C01819=1046.812,379.525,376.002,173.658,41.858,158.138
C01820=1046.820,379.771,375.961,173.664,41.863,158.140
C01821=1046.829,380.018,375.920,173.671,41.869,158.141
C01822=1046.836,380.264,375.878,173.677,41.874,158.143
C01823=1046.844,380.510,375.838,173.684,41.880,158.145
C01824=1046.852,380.757,375.797,173.690,41.885,158.146
C01825=1046.861,381.004,375.756,173.697,41.890,158.148
C01826=1046.869,381.250,375.714,173.703,41.896,158.150
C01827=1046.877,381.496,375.673,173.710,41.901,158.152
C01828=1046.885,381.743,375.632,173.716,41.907,158.154
C01829=1046.893,381.989,375.590,173.723,41.912,158.155
C01830=1046.901,382.236,375.549,173.729,41.917,158.157
C01831=1046.910,382.481,375.508,173.737,41.923,158.159
C01832=1046.918,382.728,375.467,173.743,41.929,158.161
C01833=1046.926,382.974,375.425,173.750,41.934,158.162
C01834=1046.934,383.221,375.385,173.757,41.939,158.164
C01835=1046.943,383.467,375.343,173.763,41.945,158.166
C01836=1046.950,383.714,375.302,173.770,41.950,158.168
C01837=1046.959,383.960,375.260,173.777,41.956,158.170
C01838=1046.967,384.206,375.219,173.784,41.962,158.171
C01839=1046.975,384.453,375.177,173.791,41.967,158.173
C01840=1046.984,384.699,375.136,173.797,41.973,158.175
C01841=1046.993,384.945,375.094,173.804,41.978,158.177
C01842=1047.001,385.191,375.053,173.811,41.984,158.179
C01843=1047.009,385.438,375.011,173.818,41.989,158.180
C01844=1047.018,385.684,374.969,173.825,41.995,158.182
C01845=1047.026,385.930,374.928,173.832,42.001,158.184
C01846=1047.034,386.177,374.886,173.839,42.006,158.186
C01847=1047.043,386.424,374.845,173.845,42.012,158.188
C01848=1047.051,386.669,374.803,173.852,42.018,158.190
C01849=1047.059,386.916,374.761,173.860,42.023,158.192
C01850=1047.068,387.162,374.719,173.867,42.029,158.193
C01851=1047.076,387.408,374.677,173.873,42.035,158.195
C01852=1047.085,387.655,374.635,173.880,42.041,158.197
C01853=1047.094,387.901,374.594,173.888,42.046,158.199
C01854=1047.102,388.147,374.551,173.895,42.052,158.201
C01855=1047.111,388.393,374.509,173.902,42.058,158.203
C01856=1047.120,388.639,374.468,173.909,42.064,158.205
C01857=1047.128,388.886,374.425,173.916,42.069,158.207
C01858=1047.137,389.132,374.384,173.923,42.075,158.209
C01859=1047.145,389.378,374.341,173.930,42.081,158.210
C01860=1047.158,389.751,374.278,173.941,42.090,158.213
C01861=1047.170,390.124,374.213,173.953,42.099,158.216
C01862=1047.184,390.498,374.149,173.963,42.108,158.219
C01863=1047.196,390.871,374.085,173.974,42.117,158.222
C01864=1047.205,391.117,374.042,173.981,42.123,158.224
C01865=1047.214,391.364,374.000,173.988,42.129,158.226
C01866=1047.222,391.610,373.957,173.996,42.135,158.228
C01867=1047.231,391.856,373.915,174.003,42.141,158.230
C01868=1047.240,392.102,373.872,174.011,42.147,158.232
C01869=1047.248,392.348,373.829,174.018,42.153,158.234
C01870=1047.256,392.595,373.787,174.026,42.160,158.236
C01871=1047.266,392.841,373.744,174.033,42.166,158.238
C01872=1047.274,393.087,373.701,174.041,42.172,158.240
C01873=1047.283,393.333,373.658,174.048,42.178,158.242
C01874=1047.291,393.579,373.615,174.055,42.184,158.244
C01875=1047.300,393.825,373.572,174.063,42.190,158.247
C01876=1047.308,394.071,373.531,174.071,42.196,158.249
C01877=1047.317,394.317,373.487,174.078,42.202,158.251
C01878=1047.325,394.563,373.444,174.086,42.209,158.253
C01879=1047.334,394.809,373.401,174.093,42.215,158.255
C01880=1047.343,395.055,373.359,174.100,42.221,158.257
C01881=1047.352,395.300,373.315,174.108,42.228,158.259
C01882=1047.361,395.547,373.272,174.116,42.234,158.261
C01883=1047.370,395.793,373.229,174.123,42.240,158.263
C01884=1047.378,396.039,373.186,174.131,42.247,158.265
C01885=1047.387,396.285,373.143,174.138,42.253,158.267
C01886=1047.395,396.531,373.100,174.146,42.259,158.270
C01887=1047.404,396.777,373.056,174.154,42.266,158.272
C01888=1047.413,397.024,373.013,174.161,42.272,158.274
C01889=1047.422,397.270,372.970,174.170,42.278,158.276
C01890=1047.430,397.515,372.926,174.177,42.285,158.278
C01891=1047.439,397.761,372.883,174.185,42.291,158.280
C01892=1047.448,398.007,372.839,174.193,42.298,158.282
C01893=1047.457,398.253,372.796,174.200,42.304,158.285
C01894=1047.466,398.499,372.752,174.208,42.311,158.287
C01895=1047.475,398.746,372.709,174.217,42.317,158.289
C01896=1047.483,398.991,372.665,174.224,42.324,158.291
C01897=1047.492,399.236,372.621,174.232,42.330,158.293
C01898=1047.501,399.483,372.578,174.240,42.337,158.296
C01899=1047.510,399.729,372.534,174.248,42.343,158.298
C01900=1047.520,399.975,372.490,174.256,42.350,158.300
C01901=1047.528,400.221,372.447,174.264,42.357,158.302
C01902=1047.538,400.467,372.403,174.272,42.363,158.304
C01903=1047.546,400.712,372.359,174.280,42.370,158.307
C01904=1047.556,400.959,372.315,174.288,42.377,158.309
C01905=1047.565,401.204,372.271,174.296,42.383,158.311
C01906=1047.574,401.450,372.227,174.305,42.390,158.314
C01907=1047.582,401.696,372.183,174.313,42.397,158.316
C01908=1047.591,401.943,372.139,174.320,42.404,158.318
C01909=1047.601,402.188,372.094,174.329,42.410,158.320
C01910=1047.610,402.434,372.051,174.337,42.417,158.323
C01911=1047.619,402.680,372.007,174.345,42.424,158.325
C01912=1047.627,402.925,371.962,174.354,42.431,158.327
C01913=1047.637,403.172,371.918,174.362,42.438,158.330
C01914=1047.646,403.418,371.874,174.370,42.445,158.332
C01915=1047.655,403.663,371.829,174.378,42.452,158.334
C01916=1047.669,404.055,371.758,174.392,42.463,158.338
C01917=1047.684,404.447,371.688,174.405,42.474,158.342
C01918=1047.698,404.840,371.616,174.419,42.485,158.346
C01919=1047.713,405.232,371.545,174.432,42.496,158.349
C01920=1047.722,405.478,371.501,174.440,42.503,158.352
C01921=1047.731,405.723,371.456,174.449,42.510,158.354
C01922=1047.740,405.969,371.411,174.457,42.517,158.357
C01923=1047.749,406.215,371.366,174.466,42.524,158.359
C01924=1047.759,406.460,371.321,174.474,42.532,158.362
C01925=1047.768,406.707,371.277,174.483,42.539,158.364
C01926=1047.777,406.952,371.232,174.491,42.546,158.367
C01927=1047.786,407.198,371.186,174.500,42.553,158.369
C01928=1047.796,407.444,371.141,174.510,42.560,158.372
C01929=1047.805,407.689,371.096,174.517,42.567,158.374
C01930=1047.814,407.936,371.052,174.527,42.575,158.377
C01931=1047.823,408.181,371.007,174.536,42.582,158.379
C01932=1047.833,408.427,370.962,174.544,42.589,158.381
C01933=1047.842,408.673,370.916,174.553,42.597,158.384
C01934=1047.851,408.919,370.871,174.562,42.604,158.387
C01935=1047.861,409.164,370.826,174.570,42.611,158.389
C01936=1047.870,409.409,370.780,174.580,42.619,158.392
C01937=1047.880,409.655,370.735,174.589,42.626,158.394
C01938=1047.889,409.901,370.690,174.597,42.634,158.397
C01939=1047.899,410.147,370.644,174.606,42.641,158.399
C01940=1047.908,410.393,370.599,174.615,42.648,158.402
C01941=1047.918,410.638,370.554,174.625,42.656,158.405
C01942=1047.927,410.883,370.508,174.634,42.663,158.407
C01943=1047.937,411.129,370.463,174.642,42.671,158.410
C01944=1047.947,411.375,370.417,174.651,42.679,158.412
C01945=1047.956,411.621,370.371,174.661,42.686,158.415
C01946=1047.966,411.865,370.326,174.670,42.693,158.418
C01947=1047.975,412.112,370.280,174.679,42.701,158.420
C01948=1047.985,412.357,370.234,174.688,42.708,158.423
C01949=1047.995,412.603,370.189,174.698,42.716,158.426
C01950=1048.004,412.849,370.143,174.707,42.724,158.428
C01951=1048.013,413.094,370.097,174.717,42.731,158.431
C01952=1048.024,413.340,370.051,174.726,42.739,158.434
C01953=1048.033,413.585,370.005,174.734,42.747,158.436
C01954=1048.043,413.831,369.959,174.744,42.755,158.439
C01955=1048.052,414.076,369.912,174.753,42.763,158.442
C01956=1048.062,414.322,369.866,174.763,42.770,158.445
C01957=1048.071,414.567,369.820,174.772,42.778,158.447
C01958=1048.081,414.813,369.773,174.782,42.786,158.450
C01959=1048.090,415.059,369.727,174.792,42.794,158.453
C01960=1048.101,415.304,369.681,174.802,42.802,158.456
C01961=1048.110,415.549,369.635,174.811,42.810,158.459
C01962=1048.120,415.795,369.589,174.821,42.818,158.461
C01963=1048.130,416.040,369.543,174.830,42.826,158.464
C01964=1048.140,416.286,369.495,174.840,42.833,158.467
C01965=1048.150,416.532,369.449,174.849,42.842,158.470
C01966=1048.159,416.777,369.403,174.859,42.850,158.473
C01967=1048.169,417.023,369.356,174.870,42.858,158.475
C01968=1048.179,417.268,369.309,174.879,42.866,158.478
C01969=1048.189,417.514,369.262,174.889,42.874,158.481
C01970=1048.198,417.759,369.216,174.899,42.882,158.484
C01971=1048.209,418.004,369.170,174.908,42.890,158.487
C01972=1048.225,418.404,369.093,174.925,42.904,158.492
C01973=1048.242,418.803,369.017,174.941,42.917,158.496
C01974=1048.257,419.202,368.940,174.957,42.931,158.501
C01975=1048.274,419.601,368.863,174.974,42.943,158.506
C01976=1048.283,419.846,368.816,174.984,42.952,158.509
C01977=1048.293,420.091,368.769,174.994,42.961,158.512
C01978=1048.304,420.337,368.722,175.005,42.969,158.515
C01979=1048.314,420.582,368.675,175.015,42.978,158.518
C01980=1048.323,420.827,368.627,175.026,42.986,158.521
C01981=1048.333,421.073,368.580,175.035,42.994,158.524
C01982=1048.344,421.318,368.532,175.045,43.003,158.527
C01983=1048.354,421.563,368.485,175.056,43.012,158.530
C01984=1048.364,421.809,368.438,175.066,43.020,158.533
C01985=1048.374,422.054,368.389,175.077,43.028,158.537
C01986=1048.385,422.300,368.342,175.088,43.037,158.540
C01987=1048.395,422.545,368.295,175.098,43.045,158.543
C01988=1048.405,422.789,368.247,175.109,43.054,158.546
C01989=1048.416,423.035,368.199,175.119,43.063,158.549
C01990=1048.425,423.280,368.151,175.130,43.071,158.552
C01991=1048.435,423.525,368.104,175.141,43.080,158.555
C01992=1048.447,423.770,368.055,175.151,43.089,158.558
C01993=1048.457,424.016,368.008,175.162,43.097,158.562
C01994=1048.467,424.261,367.960,175.173,43.107,158.565
C01995=1048.478,424.506,367.911,175.183,43.115,158.568
C01996=1048.488,424.751,367.864,175.194,43.124,158.571
C01997=1048.499,424.997,367.816,175.206,43.133,158.575
C01998=1048.509,425.242,367.767,175.217,43.142,158.578
C01999=1048.519,425.486,367.719,175.227,43.151,158.581
C02000=1048.530,425.732,367.670,175.238,43.160,158.584
C02001=1048.540,425.977,367.623,175.249,43.169,158.588
C02002=1048.550,426.222,367.574,175.261,43.178,158.591
C02003=1048.561,426.467,367.526,175.272,43.187,158.594
C02004=1048.571,426.712,367.477,175.283,43.195,158.597
C02005=1048.582,426.957,367.429,175.294,43.205,158.601
C02006=1048.592,427.202,367.380,175.306,43.214,158.604
C02007=1048.603,427.447,367.331,175.316,43.223,158.607
C02008=1048.613,427.693,367.282,175.328,43.233,158.611
C02009=1048.624,427.937,367.234,175.339,43.242,158.614
C02010=1048.634,428.182,367.185,175.350,43.251,158.618
C02011=1048.645,428.426,367.136,175.363,43.260,158.621
C02012=1048.656,428.672,367.087,175.374,43.269,158.625
C02013=1048.667,428.917,367.038,175.385,43.278,158.628
C02014=1048.677,429.163,366.989,175.397,43.288,158.632
C02015=1048.689,429.407,366.940,175.408,43.297,158.635
C02016=1048.699,429.652,366.891,175.420,43.306,158.638
C02017=1048.709,429.897,366.842,175.432,43.316,158.642
C02018=1048.720,430.142,366.793,175.443,43.326,158.646
C02019=1048.731,430.387,366.744,175.456,43.335,158.649
C02020=1048.741,430.631,366.694,175.467,43.345,158.653
C02021=1048.752,430.876,366.645,175.479,43.354,158.656
C02022=1048.763,431.122,366.595,175.491,43.364,158.660
C02023=1048.774,431.366,366.545,175.502,43.373,158.663
C02024=1048.785,431.611,366.496,175.515,43.383,158.667
C02025=1048.796,431.856,366.446,175.527,43.393,158.671
C02026=1048.806,432.101,366.397,175.538,43.402,158.674
C02027=1048.818,432.346,366.348,175.551,43.412,158.678
C02028=1048.826,432.556,366.304,175.561,43.421,158.681
C02029=1048.836,432.767,366.261,175.572,43.428,158.684
C02030=1048.846,432.979,366.218,175.583,43.437,158.687
C02031=1048.856,433.190,366.175,175.594,43.445,158.691
C02032=1048.865,433.402,366.132,175.604,43.454,158.694
C02033=1048.875,433.613,366.089,175.614,43.463,158.697
C02034=1048.885,433.824,366.046,175.625,43.471,158.700
C02035=1048.894,434.035,366.003,175.636,43.480,158.703
C02036=1048.905,434.280,365.952,175.648,43.489,158.707
C02037=1048.916,434.525,365.903,175.661,43.499,158.711
C02038=1048.927,434.769,365.853,175.673,43.509,158.715
C02039=1048.938,435.014,365.802,175.686,43.520,158.719
C02040=1048.950,435.258,365.752,175.699,43.529,158.723
C02041=1048.961,435.503,365.702,175.712,43.540,158.726
C02042=1048.972,435.747,365.651,175.724,43.550,158.730
C02043=1048.984,435.992,365.601,175.738,43.560,158.734
C02044=1048.995,436.237,365.550,175.750,43.570,158.738
C02045=1049.006,436.482,365.500,175.763,43.580,158.742
C02046=1049.017,436.726,365.449,175.776,43.591,158.746
C02047=1049.029,436.971,365.398,175.789,43.601,158.750
C02048=1049.040,437.215,365.348,175.802,43.611,158.754
C02049=1049.051,437.459,365.297,175.816,43.621,158.758
C02050=1049.063,437.704,365.246,175.828,43.632,158.762
C02051=1049.075,437.949,365.195,175.841,43.642,158.766
C02052=1049.086,438.193,365.144,175.854,43.653,158.770
C02053=1049.098,438.438,365.093,175.868,43.663,158.774
C02054=1049.109,438.682,365.043,175.881,43.674,158.778
C02055=1049.121,438.927,364.991,175.894,43.684,158.782
C02056=1049.133,439.171,364.940,175.908,43.695,158.786
C02057=1049.144,439.415,364.889,175.922,43.705,158.790
C02058=1049.156,439.660,364.837,175.936,43.716,158.794
C02059=1049.167,439.904,364.785,175.949,43.726,158.799
C02060=1049.179,440.149,364.734,175.963,43.737,158.803
C02061=1049.190,440.393,364.683,175.976,43.748,158.807
C02062=1049.202,440.637,364.631,175.990,43.759,158.811
C02063=1049.214,440.882,364.580,176.005,43.769,158.815
C02064=1049.226,441.126,364.528,176.018,43.780,158.820
C02065=1049.238,441.370,364.477,176.032,43.791,158.824
C02066=1049.249,441.615,364.425,176.046,43.802,158.828
C02067=1049.261,441.859,364.372,176.060,43.813,158.833
C02068=1049.273,442.103,364.321,176.074,43.824,158.837
C02069=1049.285,442.347,364.269,176.089,43.835,158.841
C02070=1049.296,442.592,364.217,176.102,43.846,158.845
C02071=1049.309,442.836,364.165,176.117,43.857,158.850
C02072=1049.321,443.080,364.113,176.131,43.868,158.854
C02073=1049.332,443.324,364.060,176.146,43.879,158.859
C02074=1049.344,443.568,364.008,176.160,43.891,158.863
C02075=1049.357,443.813,363.956,176.175,43.901,158.868
C02076=1049.368,444.057,363.903,176.189,43.913,158.872
C02077=1049.380,444.301,363.851,176.204,43.924,158.877
C02078=1049.393,444.544,363.798,176.219,43.935,158.881
C02079=1049.406,444.789,363.746,176.233,43.947,158.886
C02080=1049.417,445.033,363.693,176.248,43.958,158.890
C02081=1049.429,445.277,363.641,176.263,43.969,158.895
C02082=1049.443,445.521,363.588,176.278,43.981,158.899
C02083=1049.454,445.765,363.535,176.293,43.992,158.904
C02084=1049.467,446.008,363.483,176.308,44.004,158.909
C02085=1049.480,446.250,363.431,176.324,44.015,158.913
C02086=1049.494,446.494,363.380,176.338,44.026,158.918
C02087=1049.508,446.738,363.328,176.354,44.037,158.922
C02088=1049.524,446.976,363.279,176.368,44.047,158.926
C02089=1049.538,447.213,363.232,176.383,44.058,158.931
C02090=1049.555,447.450,363.183,176.399,44.068,158.935
C02091=1049.571,447.687,363.135,176.414,44.078,158.939
C02092=1049.589,447.926,363.089,176.429,44.088,158.944
C02093=1049.608,448.164,363.042,176.444,44.098,158.948
C02094=1049.626,448.402,362.996,176.459,44.108,158.952
C02095=1049.646,448.642,362.950,176.475,44.117,158.956
C02096=1049.666,448.886,362.904,176.490,44.127,158.961
C02097=1049.687,449.131,362.858,176.507,44.137,158.965
C02098=1049.710,449.376,362.812,176.524,44.146,158.969
C02099=1049.733,449.621,362.768,176.539,44.156,158.973
C02100=1049.757,449.867,362.724,176.556,44.165,158.977
C02101=1049.780,450.112,362.680,176.572,44.173,158.981
C02102=1049.805,450.357,362.637,176.588,44.182,158.986
C02103=1049.831,450.602,362.594,176.604,44.191,158.989
C02104=1049.518,450.631,362.293,176.605,44.282,159.016
C02105=1049.493,450.386,362.335,176.589,44.273,159.012
C02106=1049.468,450.140,362.379,176.572,44.265,159.008
C02107=1049.443,449.895,362.422,176.555,44.256,159.004
C02108=1049.419,449.650,362.467,176.539,44.247,159.000
C02109=1049.397,449.405,362.511,176.523,44.238,158.996
C02110=1049.374,449.159,362.556,176.507,44.228,158.991
C02111=1049.353,448.915,362.602,176.491,44.219,158.987
C02112=1049.332,448.670,362.648,176.474,44.209,158.983
C02113=1049.313,448.441,362.692,176.459,44.200,158.979
C02114=1049.295,448.211,362.736,176.445,44.191,158.975
C02115=1049.277,447.982,362.781,176.430,44.182,158.971
C02116=1049.259,447.753,362.826,176.415,44.172,158.967
C02117=1049.244,447.524,362.872,176.401,44.162,158.963
C02118=1049.227,447.295,362.918,176.386,44.153,158.958
C02119=1049.212,447.067,362.965,176.372,44.143,158.954
C02120=1049.198,446.839,363.011,176.357,44.133,158.950
C02121=1049.182,446.595,363.062,176.342,44.122,158.946
C02122=1049.169,446.352,363.113,176.326,44.111,158.941
C02123=1049.154,446.108,363.165,176.311,44.100,158.936
C02124=1049.142,445.865,363.216,176.296,44.089,158.932
C02125=1049.129,445.621,363.270,176.281,44.077,158.927
C02126=1049.117,445.377,363.322,176.266,44.066,158.923
C02127=1049.105,445.133,363.375,176.251,44.054,158.918
C02128=1049.092,444.890,363.427,176.236,44.044,158.914
C02129=1049.080,444.628,363.484,176.220,44.031,158.909
C02130=1049.066,444.366,363.540,176.204,44.019,158.904
C02131=1049.053,444.104,363.596,176.189,44.007,158.899
C02132=1049.040,443.842,363.653,176.173,43.995,158.894
C02133=1049.028,443.598,363.705,176.158,43.984,158.890
C02134=1049.016,443.354,363.758,176.143,43.973,158.885
C02135=1049.004,443.110,363.810,176.129,43.962,158.881
C02136=1048.992,442.866,363.862,176.114,43.951,158.876
C02137=1048.980,442.622,363.913,176.100,43.940,158.872
C02138=1048.968,442.378,363.966,176.086,43.929,158.868
C02139=1048.956,442.134,364.018,176.072,43.918,158.863
C02140=1048.944,441.889,364.070,176.057,43.907,158.859
C02141=1048.932,441.645,364.122,176.043,43.896,158.855
C02142=1048.920,441.400,364.174,176.030,43.885,158.850
C02143=1048.909,441.155,364.225,176.015,43.874,158.846
C02144=1048.896,440.912,364.278,176.001,43.864,158.842
C02145=1048.885,440.668,364.329,175.988,43.853,158.838
C02146=1048.873,440.423,364.380,175.973,43.843,158.833
C02147=1048.861,440.179,364.431,175.960,43.832,158.829
C02148=1048.850,439.934,364.483,175.946,43.821,158.825
C02149=1048.838,439.689,364.535,175.932,43.810,158.821
C02150=1048.827,439.446,364.586,175.919,43.800,158.817
C02151=1048.815,439.201,364.637,175.905,43.790,158.812
C02152=1048.803,438.957,364.689,175.891,43.779,158.808
C02153=1048.791,438.712,364.740,175.878,43.768,158.804
C02154=1048.780,438.468,364.791,175.864,43.758,158.800
C02155=1048.768,438.224,364.842,175.851,43.748,158.796
C02156=1048.757,437.979,364.893,175.837,43.737,158.792
C02157=1048.745,437.735,364.944,175.824,43.727,158.788
C02158=1048.734,437.490,364.995,175.811,43.717,158.784
C02159=1048.722,437.246,365.046,175.798,43.706,158.780
C02160=1048.711,437.001,365.097,175.784,43.696,158.776
C02161=1048.700,436.756,365.147,175.772,43.686,158.772
C02162=1048.688,436.512,365.198,175.759,43.675,158.768
C02163=1048.677,436.267,365.249,175.746,43.666,158.764
C02164=1048.666,436.023,365.299,175.733,43.655,158.760
C02165=1048.655,435.778,365.350,175.720,43.646,158.756
C02166=1048.644,435.533,365.400,175.707,43.635,158.752
C02167=1048.632,435.288,365.451,175.694,43.625,158.749
C02168=1048.620,435.044,365.500,175.681,43.616,158.745
C02169=1048.609,434.800,365.551,175.668,43.605,158.741
C02170=1048.598,434.555,365.601,175.656,43.595,158.737
C02171=1048.587,434.310,365.652,175.643,43.586,158.733
C02172=1048.575,434.066,365.702,175.631,43.576,158.730
C02173=1048.557,433.659,365.785,175.610,43.560,158.723
C02174=1048.539,433.252,365.867,175.589,43.543,158.717
C02175=1048.520,432.845,365.950,175.569,43.527,158.711
C02176=1048.502,432.438,366.033,175.549,43.511,158.705
C02177=1048.491,432.194,366.083,175.536,43.501,158.701
C02178=1048.480,431.949,366.133,175.525,43.492,158.698
C02179=1048.470,431.703,366.182,175.512,43.482,158.694
C02180=1048.458,431.459,366.232,175.500,43.472,158.690
C02181=1048.447,431.214,366.282,175.488,43.463,158.687
C02182=1048.437,430.969,366.331,175.476,43.453,158.683
C02183=1048.425,430.725,366.380,175.464,43.444,158.680
C02184=1048.414,430.479,366.430,175.452,43.434,158.676
C02185=1048.404,430.234,366.480,175.441,43.425,158.672
C02186=1048.394,429.990,366.529,175.428,43.415,158.669
C02187=1048.382,429.745,366.578,175.417,43.406,158.665
C02188=1048.372,429.500,366.627,175.405,43.397,158.662
C02189=1048.361,429.255,366.677,175.393,43.387,158.658
C02190=1048.350,429.011,366.725,175.382,43.378,158.655
C02191=1048.340,428.766,366.775,175.370,43.369,158.651
C02192=1048.329,428.520,366.823,175.359,43.360,158.648
C02193=1048.318,428.275,366.872,175.348,43.351,158.645
C02194=1048.308,428.030,366.921,175.335,43.341,158.641
C02195=1048.297,427.785,366.970,175.324,43.332,158.638
C02196=1048.287,427.540,367.019,175.312,43.323,158.634
C02197=1048.276,427.295,367.067,175.301,43.314,158.631
C02198=1048.265,427.050,367.116,175.290,43.305,158.628
C02199=1048.255,426.805,367.164,175.279,43.296,158.624
C02200=1048.244,426.560,367.213,175.268,43.287,158.621
C02201=1048.234,426.315,367.261,175.257,43.278,158.618
C02202=1048.223,426.070,367.310,175.245,43.269,158.614
C02203=1048.213,425.825,367.359,175.234,43.260,158.611
C02204=1048.202,425.580,367.407,175.223,43.251,158.608
C02205=1048.192,425.335,367.456,175.212,43.242,158.604
C02206=1048.181,425.090,367.503,175.201,43.234,158.601
C02207=1048.171,424.844,367.551,175.190,43.224,158.598
C02208=1048.161,424.599,367.600,175.179,43.216,158.595
C02209=1048.150,424.354,367.648,175.168,43.207,158.591
C02210=1048.139,424.109,367.696,175.157,43.199,158.588
C02211=1048.129,423.864,367.743,175.147,43.190,158.585
C02212=1048.119,423.618,367.792,175.136,43.181,158.582
C02213=1048.109,423.373,367.839,175.125,43.172,158.579
C02214=1048.098,423.128,367.887,175.115,43.164,158.576
C02215=1048.088,422.883,367.934,175.104,43.155,158.572
C02216=1048.078,422.637,367.983,175.093,43.147,158.569
C02217=1048.067,422.392,368.030,175.083,43.138,158.566
C02218=1048.057,422.147,368.078,175.071,43.129,158.563
C02219=1048.047,421.902,368.126,175.062,43.121,158.560
C02220=1048.036,421.657,368.173,175.051,43.112,158.557
C02221=1048.027,421.412,368.221,175.040,43.104,158.554
C02222=1048.017,421.167,368.268,175.030,43.095,158.551
C02223=1048.006,420.921,368.316,175.019,43.087,158.548
C02224=1047.996,420.676,368.363,175.009,43.078,158.545
C02225=1047.986,420.431,368.410,174.999,43.070,158.542
C02226=1047.976,420.185,368.458,174.988,43.062,158.539
C02227=1047.966,419.940,368.505,174.979,43.054,158.536
C02228=1047.956,419.695,368.552,174.968,43.045,158.532
C02229=1047.940,419.293,368.630,174.951,43.032,158.528
C02230=1047.924,418.892,368.707,174.934,43.018,158.523
C02231=1047.907,418.491,368.783,174.918,43.005,158.518
C02232=1047.891,418.089,368.861,174.902,42.991,158.513
C02233=1047.881,417.844,368.906,174.891,42.983,158.510
C02234=1047.871,417.599,368.953,174.882,42.976,158.508
C02235=1047.861,417.353,369.000,174.872,42.967,158.505
C02236=1047.850,417.108,369.047,174.862,42.959,158.502
C02237=1047.841,416.862,369.094,174.852,42.951,158.499
C02238=1047.831,416.617,369.140,174.842,42.943,158.496
C02239=1047.821,416.371,369.187,174.832,42.935,158.493
C02240=1047.811,416.125,369.233,174.823,42.927,158.490
C02241=1047.802,415.881,369.280,174.813,42.919,158.488
C02242=1047.792,415.635,369.327,174.804,42.912,158.485
C02243=1047.782,415.390,369.372,174.794,42.904,158.482
C02244=1047.772,415.144,369.419,174.784,42.896,158.479
C02245=1047.762,414.898,369.465,174.774,42.888,158.476
C02246=1047.753,414.653,369.511,174.765,42.880,158.473
C02247=1047.743,414.407,369.558,174.755,42.873,158.471
C02248=1047.734,414.162,369.604,174.746,42.865,158.468
C02249=1047.724,413.916,369.651,174.736,42.857,158.465
C02250=1047.714,413.671,369.697,174.727,42.849,158.463
C02251=1047.705,413.425,369.743,174.717,42.841,158.460
C02252=1047.694,413.180,369.789,174.708,42.834,158.457
C02253=1047.685,412.934,369.834,174.699,42.826,158.454
C02254=1047.676,412.688,369.881,174.689,42.818,158.452
C02255=1047.666,412.443,369.927,174.680,42.811,158.449
C02256=1047.656,412.197,369.972,174.670,42.803,158.446
C02257=1047.647,411.952,370.018,174.662,42.796,158.444
C02258=1047.637,411.706,370.063,174.653,42.788,158.441
C02259=1047.627,411.460,370.109,174.643,42.780,158.438
C02260=1047.618,411.214,370.155,174.634,42.773,158.436
C02261=1047.608,410.969,370.200,174.625,42.766,158.433
C02262=1047.599,410.723,370.246,174.616,42.758,158.431
C02263=1047.589,410.477,370.291,174.606,42.751,158.428
C02264=1047.580,410.232,370.337,174.598,42.744,158.425
C02265=1047.570,409.987,370.382,174.589,42.736,158.423
C02266=1047.561,409.741,370.427,174.580,42.729,158.420
C02267=1047.551,409.495,370.473,174.570,42.722,158.418
C02268=1047.542,409.249,370.518,174.561,42.714,158.415
C02269=1047.531,409.004,370.564,174.553,42.707,158.413
C02270=1047.523,408.758,370.609,174.544,42.700,158.410
C02271=1047.513,408.513,370.654,174.535,42.692,158.408
C02272=1047.504,408.267,370.699,174.527,42.685,158.405
C02273=1047.494,408.021,370.744,174.518,42.678,158.403
C02274=1047.485,407.775,370.789,174.508,42.671,158.400
C02275=1047.476,407.529,370.834,174.500,42.663,158.397
C02276=1047.467,407.283,370.879,174.491,42.656,158.395
C02277=1047.458,407.038,370.924,174.482,42.649,158.392
C02278=1047.448,406.792,370.969,174.474,42.642,158.390
C02279=1047.438,406.547,371.014,174.465,42.635,158.388
C02280=1047.430,406.300,371.059,174.457,42.628,158.385
C02281=1047.420,406.055,371.104,174.448,42.621,158.383
C02282=1047.411,405.809,371.149,174.439,42.614,158.380
C02283=1047.402,405.563,371.193,174.431,42.607,158.378
C02284=1047.393,405.318,371.238,174.422,42.599,158.375
C02285=1047.378,404.924,371.310,174.409,42.588,158.372
C02286=1047.364,404.530,371.381,174.395,42.577,158.368
C02287=1047.349,404.135,371.453,174.381,42.566,158.364
C02288=1047.335,403.741,371.524,174.368,42.555,158.360
C02289=1047.325,403.495,371.569,174.360,42.548,158.358
C02290=1047.316,403.249,371.613,174.351,42.541,158.355
C02291=1047.307,403.004,371.657,174.343,42.534,158.353
C02292=1047.298,402.757,371.701,174.334,42.528,158.351
C02293=1047.289,402.511,371.746,174.326,42.521,158.349
C02294=1047.280,402.266,371.790,174.318,42.514,158.346
C02295=1047.271,402.020,371.834,174.310,42.508,158.344
C02296=1047.262,401.774,371.879,174.302,42.501,158.342
C02297=1047.253,401.528,371.923,174.294,42.494,158.339
C02298=1047.244,401.282,371.967,174.285,42.487,158.337
C02299=1047.235,401.037,372.010,174.277,42.481,158.335
C02300=1047.226,400.790,372.054,174.270,42.474,158.333
C02301=1047.217,400.544,372.098,174.261,42.467,158.330
C02302=1047.208,400.298,372.142,174.253,42.461,158.328
C02303=1047.198,400.052,372.186,174.245,42.454,158.326
C02304=1047.189,399.807,372.230,174.236,42.448,158.324
C02305=1047.182,399.560,372.273,174.229,42.441,158.321
C02306=1047.172,399.314,372.317,174.221,42.435,158.319
C02307=1047.163,399.069,372.361,174.213,42.428,158.317
C02308=1047.154,398.822,372.404,174.204,42.421,158.315
C02309=1047.145,398.577,372.448,174.197,42.415,158.312
C02310=1047.136,398.330,372.492,174.189,42.409,158.310
C02311=1047.127,398.084,372.535,174.182,42.402,158.308
C02312=1047.119,397.838,372.578,174.174,42.396,158.306
C02313=1047.110,397.593,372.622,174.165,42.389,158.304
C02314=1047.101,397.346,372.665,174.157,42.383,158.302
C02315=1047.092,397.101,372.709,174.150,42.376,158.299
C02316=1047.084,396.855,372.752,174.142,42.370,158.297
C02317=1047.075,396.609,372.795,174.135,42.364,158.295
C02318=1047.066,396.363,372.839,174.127,42.357,158.293
C02319=1047.057,396.117,372.882,174.119,42.351,158.291
C02320=1047.048,395.871,372.925,174.111,42.345,158.289
C02321=1047.040,395.625,372.968,174.103,42.339,158.287
C02322=1047.031,395.379,373.011,174.096,42.332,158.285
C02323=1047.022,395.132,373.055,174.088,42.326,158.283
C02324=1047.013,394.886,373.098,174.080,42.320,158.280
C02325=1047.004,394.641,373.140,174.073,42.314,158.278
C02326=1046.995,394.395,373.183,174.066,42.308,158.276
C02327=1046.987,394.149,373.226,174.058,42.301,158.274
C02328=1046.978,393.903,373.269,174.050,42.295,158.272
C02329=1046.969,393.657,373.312,174.043,42.289,158.270
C02330=1046.961,393.411,373.355,174.035,42.283,158.268
C02331=1046.953,393.164,373.397,174.028,42.277,158.266
C02332=1046.944,392.918,373.440,174.020,42.271,158.264
C02333=1046.936,392.672,373.483,174.013,42.265,158.262
C02334=1046.926,392.426,373.526,174.005,42.259,158.260
C02335=1046.918,392.180,373.569,173.998,42.252,158.258
C02336=1046.910,391.933,373.611,173.991,42.246,158.256
C02337=1046.901,391.687,373.654,173.983,42.240,158.254
C02338=1046.892,391.441,373.696,173.976,42.234,158.252
C02339=1046.884,391.195,373.739,173.968,42.229,158.250
C02340=1046.874,390.949,373.781,173.961,42.223,158.248
C02341=1046.862,390.573,373.846,173.950,42.214,158.245
C02342=1046.849,390.198,373.910,173.939,42.205,158.242
C02343=1046.835,389.823,373.975,173.928,42.196,158.239
C02344=1046.823,389.448,374.039,173.917,42.186,158.236
C02345=1046.814,389.202,374.082,173.910,42.181,158.234
C02346=1046.806,388.955,374.124,173.903,42.175,158.232
C02347=1046.797,388.709,374.166,173.896,42.169,158.230
C02348=1046.788,388.464,374.208,173.888,42.163,158.228
C02349=1046.780,388.217,374.250,173.881,42.158,158.226
C02350=1046.771,387.971,374.292,173.875,42.152,158.225
C02351=1046.763,387.724,374.334,173.867,42.146,158.223
C02352=1046.755,387.478,374.376,173.860,42.141,158.221
C02353=1046.746,387.232,374.417,173.853,42.135,158.219
C02354=1046.738,386.985,374.460,173.846,42.130,158.217
C02355=1046.729,386.739,374.501,173.839,42.123,158.215
C02356=1046.720,386.493,374.543,173.832,42.118,158.213
C02357=1046.712,386.247,374.585,173.825,42.112,158.211
C02358=1046.703,386.000,374.627,173.818,42.107,158.210
C02359=1046.695,385.755,374.668,173.811,42.101,158.208
C02360=1046.687,385.507,374.710,173.804,42.096,158.206
C02361=1046.678,385.261,374.751,173.797,42.090,158.204
C02362=1046.670,385.015,374.793,173.790,42.085,158.202
C02363=1046.662,384.769,374.835,173.784,42.079,158.200
C02364=1046.653,384.523,374.876,173.776,42.074,158.199
C02365=1046.645,384.276,374.917,173.769,42.068,158.197
C02366=1046.636,384.030,374.959,173.763,42.062,158.195
C02367=1046.628,383.784,375.001,173.756,42.057,158.193
C02368=1046.620,383.537,375.042,173.749,42.051,158.191
C02369=1046.611,383.291,375.083,173.743,42.046,158.190
C02370=1046.604,383.044,375.125,173.735,42.041,158.188
C02371=1046.595,382.798,375.166,173.729,42.035,158.186
C02372=1046.587,382.552,375.207,173.722,42.029,158.184
C02373=1046.579,382.305,375.249,173.715,42.024,158.183
C02374=1046.571,382.059,375.290,173.709,42.019,158.181
C02375=1046.562,381.813,375.331,173.702,42.013,158.179
C02376=1046.554,381.566,375.372,173.696,42.008,158.177
C02377=1046.546,381.320,375.413,173.689,42.003,158.175
C02378=1046.537,381.073,375.455,173.682,41.997,158.174
C02379=1046.529,380.827,375.496,173.675,41.992,158.172
C02380=1046.521,380.581,375.536,173.668,41.986,158.170
C02381=1046.514,380.335,375.578,173.662,41.981,158.168
C02382=1046.505,380.088,375.619,173.655,41.976,158.167
C02383=1046.497,379.841,375.660,173.649,41.970,158.165
C02384=1046.489,379.595,375.701,173.642,41.965,158.163
C02385=1046.481,379.348,375.742,173.636,41.960,158.162
C02386=1046.473,379.101,375.783,173.629,41.955,158.160
C02387=1046.465,378.855,375.824,173.623,41.950,158.158
C02388=1046.457,378.608,375.865,173.616,41.945,158.157
C02389=1046.449,378.362,375.905,173.610,41.939,158.155
C02390=1046.441,378.116,375.946,173.603,41.934,158.153
C02391=1046.432,377.870,375.986,173.597,41.929,158.151
C02392=1046.423,377.623,376.027,173.590,41.924,158.150
C02393=1046.415,377.376,376.067,173.584,41.919,158.148
C02394=1046.407,377.130,376.108,173.578,41.913,158.147
C02395=1046.399,376.883,376.148,173.571,41.908,158.145
C02396=1046.391,376.637,376.189,173.565,41.903,158.143
C02397=1046.380,376.295,376.245,173.556,41.896,158.141
C02398=1046.368,375.953,376.301,173.547,41.889,158.139
C02399=1046.357,375.610,376.357,173.538,41.882,158.136
C02400=1046.347,375.269,376.414,173.529,41.875,158.134
C02401=1046.338,375.022,376.453,173.523,41.870,158.133
C02402=1046.330,374.775,376.494,173.518,41.865,158.131
C02403=1046.322,374.528,376.534,173.511,41.861,158.129
C02404=1046.314,374.282,376.574,173.505,41.855,158.128
C02405=1046.306,374.036,376.615,173.499,41.850,158.126
C02406=1046.298,373.789,376.655,173.492,41.845,158.124
C02407=1046.291,373.542,376.695,173.486,41.841,158.123
C02408=1046.283,373.295,376.736,173.480,41.835,158.121
C02409=1046.275,373.049,376.776,173.473,41.830,158.120
C02410=1046.267,372.802,376.816,173.468,41.826,158.118
C02411=1046.259,372.556,376.855,173.462,41.821,158.117
C02412=1046.251,372.310,376.895,173.455,41.816,158.115
C02413=1046.243,372.063,376.936,173.449,41.811,158.113
C02414=1046.236,371.816,376.976,173.443,41.806,158.112
C02415=1046.228,371.569,377.016,173.437,41.801,158.110
C02416=1046.220,371.322,377.055,173.431,41.797,158.109
C02417=1046.212,371.076,377.096,173.425,41.791,158.107
C02418=1046.204,370.830,377.135,173.419,41.787,158.106
C02419=1046.196,370.583,377.175,173.413,41.782,158.104
C02420=1046.187,370.336,377.215,173.406,41.777,158.103
C02421=1046.180,370.089,377.255,173.400,41.773,158.101
C02422=1046.173,369.843,377.294,173.395,41.768,158.100
C02423=1046.164,369.596,377.333,173.389,41.763,158.098
C02424=1046.156,369.350,377.373,173.383,41.758,158.097
C02425=1046.148,369.102,377.412,173.376,41.754,158.095
C02426=1046.141,368.855,377.452,173.371,41.749,158.094
C02427=1046.132,368.609,377.491,173.365,41.744,158.092
C02428=1046.125,368.363,377.531,173.359,41.740,158.091
C02429=1046.117,368.116,377.571,173.353,41.735,158.089
C02430=1046.109,367.869,377.610,173.347,41.731,158.088
C02431=1046.101,367.622,377.649,173.341,41.726,158.086
C02432=1046.094,367.376,377.688,173.335,41.721,158.085
C02433=1046.086,367.129,377.728,173.330,41.717,158.083
C02434=1046.077,366.882,377.767,173.324,41.712,158.082
C02435=1046.070,366.635,377.807,173.318,41.707,158.080
C02436=1046.062,366.389,377.846,173.312,41.703,158.079
C02437=1046.054,366.142,377.885,173.306,41.698,158.078
C02438=1046.046,365.895,377.924,173.300,41.694,158.076
C02439=1046.039,365.648,377.964,173.294,41.689,158.075
C02440=1046.031,365.401,378.002,173.289,41.684,158.073
C02441=1046.024,365.155,378.042,173.283,41.680,158.072
C02442=1046.016,364.908,378.080,173.277,41.675,158.070
C02443=1046.008,364.661,378.120,173.272,41.671,158.069
C02444=1046.000,364.414,378.159,173.266,41.666,158.067
C02445=1045.993,364.167,378.198,173.260,41.662,158.066
C02446=1045.985,363.921,378.237,173.254,41.657,158.065
C02447=1045.978,363.673,378.276,173.249,41.653,158.063
C02448=1045.970,363.428,378.315,173.243,41.648,158.062
C02449=1045.962,363.180,378.354,173.238,41.644,158.060
C02450=1045.955,362.933,378.392,173.232,41.639,158.059
C02451=1045.947,362.687,378.432,173.226,41.635,158.058
C02452=1045.940,362.440,378.470,173.221,41.630,158.056
C02453=1045.929,362.117,378.522,173.213,41.625,158.054
C02454=1045.919,361.795,378.572,173.205,41.619,158.052
C02455=1045.910,361.471,378.622,173.198,41.613,158.051
C02456=1045.899,361.149,378.673,173.191,41.608,158.049
C02457=1045.892,360.902,378.712,173.186,41.603,158.048
C02458=1045.884,360.655,378.750,173.180,41.599,158.046
C02459=1045.876,360.408,378.789,173.175,41.595,158.045
C02460=1045.869,360.161,378.827,173.169,41.590,158.043
C02461=1045.860,359.914,378.866,173.163,41.586,158.042
C02462=1045.854,359.667,378.904,173.158,41.582,158.041
C02463=1045.846,359.420,378.943,173.152,41.578,158.040
C02464=1045.838,359.174,378.981,173.147,41.573,158.038
C02465=1045.830,358.927,379.019,173.141,41.569,158.037
C02466=1045.822,358.680,379.058,173.136,41.565,158.035
C02467=1045.816,358.433,379.096,173.130,41.561,158.034
C02468=1045.808,358.186,379.134,173.124,41.556,158.033
C02469=1045.800,357.939,379.173,173.119,41.552,158.031
C02470=1045.793,357.692,379.211,173.113,41.548,158.030
C02471=1045.785,357.445,379.249,173.109,41.544,158.029
C02472=1045.777,357.198,379.287,173.103,41.539,158.028
C02473=1045.770,356.951,379.326,173.098,41.535,158.026
C02474=1045.763,356.704,379.364,173.093,41.531,158.025
C02475=1045.755,356.457,379.402,173.087,41.527,158.024
C02476=1045.747,356.210,379.441,173.082,41.523,158.022
C02477=1045.739,355.963,379.478,173.076,41.519,158.021
C02478=1045.732,355.717,379.516,173.071,41.515,158.020
C02479=1045.724,355.469,379.554,173.066,41.511,158.018
C02480=1045.716,355.223,379.592,173.061,41.506,158.017
C02481=1045.709,354.975,379.629,173.055,41.502,158.016
C02482=1045.702,354.729,379.668,173.050,41.498,158.015
C02483=1045.694,354.481,379.706,173.044,41.494,158.013
C02484=1045.687,354.234,379.743,173.039,41.490,158.012
C02485=1045.679,353.987,379.781,173.034,41.486,158.011
C02486=1045.672,353.740,379.819,173.029,41.482,158.010
C02487=1045.665,353.493,379.856,173.023,41.478,158.008
C02488=1045.657,353.247,379.895,173.018,41.474,158.007
C02489=1045.650,353.000,379.932,173.012,41.470,158.006
C02490=1045.642,352.752,379.970,173.008,41.465,158.004
C02491=1045.634,352.505,380.008,173.003,41.462,158.003
C02492=1045.627,352.258,380.046,172.997,41.458,158.002
C02493=1045.620,352.011,380.083,172.992,41.454,158.001
C02494=1045.613,351.764,380.121,172.987,41.450,158.000
C02495=1045.605,351.517,380.158,172.982,41.446,157.998
C02496=1045.598,351.270,380.197,172.976,41.442,157.997
C02497=1045.591,351.023,380.234,172.971,41.438,157.996
C02498=1045.583,350.776,380.271,172.967,41.434,157.995
C02499=1045.575,350.529,380.309,172.961,41.430,157.993
C02500=1045.568,350.282,380.346,172.956,41.426,157.992
C02501=1045.561,350.035,380.384,172.951,41.422,157.991
C02502=1045.554,349.788,380.421,172.946,41.418,157.990
C02503=1045.546,349.541,380.458,172.941,41.414,157.989
C02504=1045.538,349.294,380.496,172.935,41.411,157.987
C02505=1045.531,349.046,380.533,172.931,41.406,157.986
C02506=1045.523,348.799,380.569,172.926,41.403,157.985
C02507=1045.516,348.552,380.607,172.920,41.399,157.984
C02508=1045.509,348.305,380.644,172.916,41.395,157.983
C02509=1045.499,347.988,380.692,172.909,41.390,157.981
C02510=1045.490,347.670,380.740,172.902,41.385,157.980
C02511=1045.480,347.353,380.787,172.896,41.381,157.978
C02512=1045.471,347.036,380.835,172.890,41.375,157.977
C02513=1045.463,346.790,380.872,172.885,41.372,157.975
C02514=1045.456,346.543,380.909,172.879,41.368,157.974
C02515=1045.449,346.295,380.946,172.875,41.364,157.973
C02516=1045.441,346.048,380.983,172.870,41.360,157.972
C02517=1045.434,345.801,381.021,172.865,41.357,157.971
C02518=1045.427,345.553,381.057,172.860,41.353,157.970
C02519=1045.419,345.306,381.094,172.855,41.349,157.968
C02520=1045.412,345.059,381.131,172.850,41.345,157.967
C02521=1045.405,344.812,381.168,172.845,41.342,157.966
C02522=1045.398,344.565,381.205,172.841,41.338,157.965
C02523=1045.391,344.318,381.242,172.835,41.334,157.964
C02524=1045.383,344.070,381.278,172.830,41.331,157.963
C02525=1045.376,343.823,381.316,172.826,41.327,157.962
C02526=1045.369,343.576,381.352,172.820,41.323,157.960
C02527=1045.361,343.329,381.389,172.816,41.319,157.959
C02528=1045.354,343.082,381.425,172.811,41.315,157.958
C02529=1045.347,342.834,381.462,172.807,41.312,157.957
C02530=1045.340,342.587,381.499,172.801,41.308,157.956
C02531=1045.332,342.340,381.536,172.796,41.305,157.955
C02532=1045.326,342.092,381.572,172.792,41.301,157.954
C02533=1045.318,341.855,381.607,172.787,41.298,157.953
C02534=1045.312,341.617,381.642,172.782,41.294,157.952
C02535=1045.304,341.379,381.678,172.778,41.290,157.950
C02536=1045.297,341.142,381.713,172.773,41.287,157.949
C02537=1045.290,340.904,381.748,172.769,41.284,157.948
C02538=1045.283,340.667,381.783,172.764,41.280,157.947
C02539=1045.276,340.428,381.818,172.759,41.277,157.946
C02540=1045.269,340.191,381.853,172.755,41.273,157.945
C02541=1045.262,339.943,381.890,172.750,41.270,157.944
C02542=1045.255,339.696,381.925,172.746,41.266,157.943
C02543=1045.247,339.449,381.962,172.741,41.263,157.942
C02544=1045.240,339.201,381.998,172.736,41.259,157.941
C02545=1045.233,338.955,382.034,172.731,41.256,157.940
C02546=1045.225,338.707,382.071,172.727,41.252,157.939
C02547=1045.219,338.460,382.107,172.722,41.249,157.938
C02548=1045.211,338.213,382.143,172.717,41.245,157.937
C02549=1045.204,337.965,382.179,172.712,41.241,157.935
C02550=1045.197,337.718,382.215,172.708,41.238,157.934
C02551=1045.190,337.470,382.251,172.703,41.235,157.933
C02552=1045.183,337.223,382.287,172.699,41.231,157.932
C02553=1045.175,336.976,382.323,172.694,41.228,157.931
C02554=1045.169,336.729,382.360,172.689,41.224,157.930
C02555=1045.161,336.481,382.396,172.685,41.220,157.929
C02556=1045.154,336.235,382.432,172.680,41.217,157.928
C02557=1045.147,335.987,382.467,172.676,41.214,157.927
C02558=1045.140,335.739,382.504,172.670,41.210,157.926
C02559=1045.133,335.492,382.540,172.666,41.207,157.925
C02560=1045.126,335.245,382.575,172.662,41.203,157.924
C02561=1045.118,334.997,382.611,172.657,41.200,157.923
C02562=1045.111,334.750,382.647,172.653,41.196,157.922
C02563=1045.104,334.502,382.683,172.648,41.193,157.921
C02564=1045.097,334.256,382.719,172.643,41.190,157.920
C02565=1045.087,333.916,382.768,172.637,41.186,157.918
C02566=1045.077,333.576,382.817,172.631,41.181,157.917
C02567=1045.068,333.236,382.866,172.625,41.176,157.916
C02568=1045.058,332.896,382.915,172.618,41.171,157.914
C02569=1045.050,332.649,382.951,172.614,41.168,157.913
C02570=1045.043,332.401,382.986,172.610,41.165,157.912
C02571=1045.036,332.154,383.022,172.605,41.161,157.911
C02572=1045.029,331.906,383.057,172.601,41.158,157.910
C02573=1045.022,331.660,383.093,172.596,41.155,157.909
C02574=1045.015,331.412,383.128,172.591,41.152,157.908
C02575=1045.008,331.164,383.164,172.587,41.148,157.907
C02576=1045.001,330.917,383.200,172.583,41.145,157.906
C02577=1044.994,330.670,383.235,172.578,41.142,157.905
C02578=1044.986,330.422,383.270,172.574,41.138,157.904
C02579=1044.979,330.175,383.306,172.570,41.135,157.903
C02580=1044.973,329.928,383.341,172.565,41.132,157.902
C02581=1044.965,329.680,383.377,172.561,41.128,157.901
C02582=1044.958,329.432,383.412,172.557,41.125,157.900
C02583=1044.951,329.186,383.448,172.552,41.122,157.899
C02584=1044.944,328.938,383.483,172.547,41.118,157.898
C02585=1044.936,328.691,383.518,172.543,41.115,157.897
C02586=1044.930,328.443,383.553,172.539,41.112,157.896
C02587=1044.923,328.196,383.588,172.534,41.109,157.895
C02588=1044.915,327.948,383.623,172.530,41.106,157.894
C02589=1044.908,327.701,383.658,172.526,41.103,157.893
C02590=1044.901,327.454,383.693,172.521,41.100,157.892
C02591=1044.893,327.206,383.728,172.517,41.096,157.891
C02592=1044.886,326.958,383.763,172.513,41.093,157.891
C02593=1044.879,326.711,383.798,172.508,41.090,157.890
C02594=1044.872,326.464,383.833,172.504,41.087,157.889
C02595=1044.864,326.216,383.868,172.500,41.084,157.888
C02596=1044.857,325.969,383.903,172.495,41.081,157.887
C02597=1044.851,325.721,383.937,172.490,41.078,157.886
C02598=1044.843,325.474,383.972,172.487,41.075,157.885
C02599=1044.837,325.226,384.007,172.482,41.072,157.884
C02600=1044.828,324.979,384.042,172.478,41.069,157.883
C02601=1044.822,324.731,384.077,172.473,41.066,157.882
C02602=1044.815,324.484,384.112,172.469,41.062,157.881
C02603=1044.808,324.236,384.146,172.465,41.059,157.880
C02604=1044.801,323.989,384.181,172.461,41.056,157.879
C02605=1044.793,323.742,384.216,172.457,41.053,157.878
C02606=1044.787,323.494,384.251,172.452,41.050,157.877
C02607=1044.779,323.246,384.285,172.448,41.047,157.877
C02608=1044.772,322.999,384.320,172.444,41.044,157.876
C02609=1044.765,322.751,384.355,172.440,41.041,157.875
C02610=1044.758,322.504,384.389,172.436,41.038,157.874
C02611=1044.751,322.256,384.424,172.431,41.035,157.873
C02612=1044.744,322.009,384.459,172.427,41.031,157.872
C02613=1044.737,321.761,384.493,172.423,41.029,157.871
C02614=1044.730,321.514,384.528,172.419,41.026,157.870
C02615=1044.723,321.266,384.562,172.415,41.022,157.869
C02616=1044.716,321.019,384.597,172.411,41.019,157.868
C02617=1044.709,320.771,384.631,172.406,41.017,157.867
C02618=1044.702,320.524,384.666,172.402,41.014,157.867
C02619=1044.695,320.276,384.700,172.398,41.010,157.866
C02620=1044.689,320.029,384.735,172.394,41.007,157.865
C02621=1044.679,319.703,384.781,172.389,41.003,157.864
C02622=1044.670,319.377,384.826,172.383,40.999,157.862
C02623=1044.661,319.051,384.871,172.378,40.996,157.861
C02624=1044.652,318.725,384.916,172.373,40.991,157.860
C02625=1044.645,318.479,384.950,172.369,40.989,157.859
C02626=1044.639,318.231,384.985,172.364,40.986,157.858
C02627=1044.631,317.983,385.019,172.360,40.982,157.857
C02628=1044.625,317.736,385.054,172.356,40.980,157.856
C02629=1044.617,317.488,385.088,172.352,40.977,157.856
C02630=1044.611,317.240,385.122,172.348,40.973,157.855
C02631=1044.603,316.993,385.157,172.344,40.971,157.854
C02632=1044.597,316.745,385.191,172.340,40.968,157.853
C02633=1044.590,316.498,385.224,172.336,40.964,157.852
C02634=1044.584,316.250,385.259,172.332,40.962,157.851
C02635=1044.576,316.003,385.293,172.328,40.959,157.850
C02636=1044.570,315.755,385.328,172.324,40.956,157.849
C02637=1044.563,315.508,385.362,172.320,40.953,157.848
C02638=1044.557,315.260,385.396,172.316,40.950,157.848
C02639=1044.550,315.013,385.430,172.312,40.947,157.847
C02640=1044.543,314.765,385.465,172.308,40.944,157.846
C02641=1044.536,314.518,385.499,172.304,40.941,157.845
C02642=1044.530,314.270,385.533,172.300,40.938,157.844
C02643=1044.523,314.023,385.566,172.296,40.935,157.843
C02644=1044.516,313.775,385.601,172.292,40.932,157.842
C02645=1044.510,313.528,385.634,172.288,40.929,157.841
C02646=1044.503,313.280,385.669,172.284,40.926,157.841
C02647=1044.496,313.032,385.703,172.280,40.923,157.840
C02648=1044.490,312.785,385.737,172.277,40.920,157.839
C02649=1044.483,312.537,385.770,172.272,40.917,157.838
C02650=1044.476,312.290,385.804,172.269,40.915,157.837
C02651=1044.468,312.042,385.838,172.265,40.912,157.836
C02652=1044.462,311.795,385.871,172.261,40.909,157.836
C02653=1044.455,311.547,385.905,172.257,40.906,157.835
C02654=1044.448,311.299,385.938,172.253,40.903,157.834
C02655=1044.441,311.051,385.972,172.248,40.901,157.833
C02656=1044.434,310.804,386.006,172.244,40.898,157.832
C02657=1044.426,310.557,386.039,172.240,40.895,157.831
C02658=1044.419,310.309,386.072,172.236,40.892,157.831
C02659=1044.412,310.061,386.106,172.233,40.890,157.830
C02660=1044.405,309.814,386.139,172.229,40.887,157.829
C02661=1044.398,309.566,386.172,172.225,40.885,157.828
C02662=1044.391,309.318,386.206,172.221,40.881,157.827
C02663=1044.385,309.071,386.240,172.218,40.879,157.827
C02664=1044.378,308.823,386.273,172.214,40.876,157.826
C02665=1044.371,308.575,386.307,172.210,40.873,157.825
C02666=1044.363,308.328,386.340,172.206,40.871,157.824
C02667=1044.356,308.080,386.373,172.202,40.868,157.823
C02668=1044.349,307.832,386.406,172.198,40.865,157.822
C02669=1044.343,307.585,386.439,172.195,40.862,157.822
C02670=1044.336,307.337,386.473,172.191,40.860,157.821
C02671=1044.329,307.090,386.506,172.187,40.857,157.820
C02672=1044.322,306.842,386.540,172.183,40.854,157.819
C02673=1044.315,306.595,386.572,172.179,40.852,157.819
C02674=1044.308,306.347,386.606,172.175,40.849,157.818
C02675=1044.301,306.099,386.639,172.171,40.846,157.817
C02676=1044.294,305.852,386.672,172.168,40.844,157.816
C02677=1044.285,305.530,386.715,172.162,40.840,157.815
C02678=1044.276,305.209,386.759,172.158,40.836,157.814
C02679=1044.268,304.888,386.801,172.153,40.833,157.813
C02680=1044.259,304.567,386.845,172.148,40.829,157.812
C02681=1044.253,304.319,386.877,172.144,40.827,157.811
C02682=1044.245,304.071,386.910,172.140,40.824,157.810
C02683=1044.238,303.824,386.943,172.136,40.822,157.810
C02684=1044.231,303.576,386.976,172.134,40.819,157.809
C02685=1044.225,303.328,387.009,172.130,40.816,157.808
C02686=1044.218,303.081,387.043,172.126,40.813,157.807
C02687=1044.212,302.833,387.076,172.122,40.811,157.807
C02688=1044.205,302.586,387.108,172.118,40.808,157.806
C02689=1044.198,302.338,387.141,172.114,40.806,157.805
C02690=1044.191,302.091,387.174,172.111,40.803,157.804
C02691=1044.184,301.842,387.207,172.108,40.800,157.803
C02692=1044.178,301.595,387.240,172.104,40.797,157.803
C02693=1044.171,301.347,387.272,172.100,40.795,157.802
C02694=1044.164,301.099,387.305,172.096,40.792,157.801
C02695=1044.157,300.852,387.339,172.092,40.790,157.800
C02696=1044.151,300.604,387.372,172.089,40.787,157.800
C02697=1044.144,300.356,387.405,172.086,40.784,157.799
C02698=1044.137,300.109,387.437,172.082,40.781,157.798
C02699=1044.130,299.861,387.470,172.078,40.779,157.797
C02700=1044.124,299.613,387.503,172.074,40.776,157.796
C02701=1044.118,299.365,387.536,172.071,40.773,157.796
C02702=1044.111,299.117,387.569,172.067,40.771,157.795
C02703=1044.104,298.870,387.601,172.064,40.768,157.794
C02704=1044.098,298.622,387.634,172.060,40.765,157.793
C02705=1044.091,298.375,387.666,172.056,40.763,157.793
C02706=1044.084,298.126,387.699,172.053,40.760,157.792
C02707=1044.078,297.879,387.732,172.049,40.757,157.791
C02708=1044.071,297.632,387.764,172.045,40.755,157.790
C02709=1044.065,297.384,387.797,172.041,40.752,157.789
C02710=1044.058,297.136,387.830,172.039,40.750,157.789
C02711=1044.052,296.888,387.863,172.035,40.747,157.788
C02712=1044.045,296.640,387.896,172.031,40.745,157.787
C02713=1044.038,296.393,387.928,172.027,40.742,157.787
C02714=1044.031,296.145,387.961,172.024,40.739,157.786
C02715=1044.025,295.897,387.994,172.021,40.737,157.785
C02716=1044.019,295.649,388.026,172.017,40.734,157.784
C02717=1044.012,295.402,388.058,172.013,40.731,157.783
C02718=1044.004,295.154,388.090,172.010,40.729,157.783
C02719=1043.998,294.906,388.123,172.006,40.726,157.782
C02720=1043.991,294.658,388.154,172.003,40.724,157.781
C02721=1043.985,294.411,388.187,172.000,40.721,157.781
C02722=1043.978,294.163,388.219,171.996,40.719,157.780
C02723=1043.971,293.915,388.252,171.992,40.716,157.779
C02724=1043.964,293.667,388.284,171.988,40.714,157.778
C02725=1043.958,293.420,388.317,171.986,40.711,157.778
C02726=1043.951,293.172,388.348,171.982,40.709,157.777
C02727=1043.944,292.924,388.381,171.978,40.706,157.776
C02728=1043.938,292.676,388.413,171.974,40.704,157.776
C02729=1043.931,292.428,388.445,171.972,40.701,157.775
C02730=1043.924,292.180,388.476,171.968,40.699,157.774
C02731=1043.918,291.933,388.509,171.964,40.696,157.773
C02732=1043.911,291.685,388.540,171.961,40.694,157.773
C02733=1043.903,291.380,388.581,171.956,40.691,157.772
C02734=1043.894,291.075,388.619,171.952,40.688,157.771
C02735=1043.886,290.771,388.659,171.948,40.685,157.770
C02736=1043.877,290.465,388.698,171.943,40.681,157.769
C02737=1043.871,290.218,388.731,171.941,40.679,157.768
C02738=1043.864,289.970,388.762,171.937,40.677,157.768
C02739=1043.858,289.722,388.794,171.933,40.674,157.767
C02740=1043.851,289.475,388.826,171.930,40.672,157.766
C02741=1043.845,289.226,388.858,171.927,40.669,157.766
C02742=1043.838,288.979,388.889,171.923,40.667,157.765
C02743=1043.831,288.731,388.922,171.920,40.664,157.764
C02744=1043.824,288.483,388.953,171.916,40.662,157.764
C02745=1043.818,288.234,388.985,171.914,40.659,157.763
C02746=1043.810,287.987,389.017,171.910,40.657,157.762
C02747=1043.804,287.739,389.049,171.906,40.655,157.761
C02748=1043.797,287.491,389.080,171.903,40.652,157.761
C02749=1043.791,287.243,389.112,171.900,40.650,157.760
C02750=1043.784,286.996,389.145,171.896,40.647,157.759
C02751=1043.777,286.748,389.176,171.893,40.645,157.759
C02752=1043.771,286.500,389.207,171.889,40.642,157.758
C02753=1043.764,286.252,389.239,171.886,40.640,157.757
C02754=1043.757,286.004,389.270,171.883,40.638,157.757
C02755=1043.750,285.756,389.302,171.879,40.635,157.756
C02756=1043.744,285.508,389.333,171.876,40.633,157.755
C02757=1043.737,285.261,389.365,171.873,40.630,157.754
C02758=1043.730,285.013,389.396,171.869,40.628,157.754
C02759=1043.723,284.765,389.428,171.866,40.626,157.753
C02760=1043.716,284.517,389.460,171.862,40.624,157.752
C02761=1043.710,284.270,389.491,171.860,40.621,157.752
C02762=1043.703,284.022,389.522,171.856,40.619,157.751
C02763=1043.696,283.774,389.554,171.852,40.617,157.750
C02764=1043.690,283.526,389.585,171.849,40.614,157.750
C02765=1043.683,283.278,389.617,171.846,40.612,157.749
C02766=1043.676,283.030,389.648,171.843,40.609,157.748
C02767=1043.670,282.782,389.679,171.839,40.607,157.748
C02768=1043.663,282.534,389.710,171.837,40.605,157.747
C02769=1043.656,282.286,389.742,171.833,40.602,157.746
C02770=1043.650,282.038,389.773,171.829,40.600,157.746
C02771=1043.643,281.790,389.805,171.826,40.597,157.745
C02772=1043.636,281.542,389.836,171.823,40.595,157.744
C02773=1043.629,281.294,389.867,171.820,40.593,157.744
C02774=1043.623,281.046,389.899,171.816,40.590,157.743
C02775=1043.616,280.798,389.930,171.814,40.588,157.742
C02776=1043.609,280.550,389.961,171.810,40.585,157.742
C02777=1043.603,280.302,389.992,171.807,40.583,157.741
C02778=1043.597,280.055,390.024,171.803,40.581,157.740
C02779=1043.590,279.807,390.055,171.801,40.578,157.740
C02780=1043.583,279.559,390.086,171.797,40.576,157.739
C02781=1043.577,279.310,390.117,171.794,40.574,157.738
C02782=1043.570,279.062,390.149,171.790,40.571,157.738
C02783=1043.563,278.815,390.180,171.788,40.569,157.737
C02784=1043.557,278.566,390.211,171.784,40.567,157.736
C02785=1043.551,278.319,390.242,171.781,40.564,157.736
C02786=1043.543,278.071,390.273,171.778,40.562,157.735
C02787=1043.537,277.823,390.303,171.775,40.560,157.734
C02788=1043.530,277.575,390.335,171.771,40.558,157.734
C02789=1043.522,277.282,390.371,171.767,40.554,157.733
C02790=1043.515,276.989,390.408,171.764,40.552,157.732
C02791=1043.506,276.696,390.444,171.760,40.549,157.731
C02792=1043.499,276.403,390.481,171.756,40.546,157.731
C02793=1043.491,276.154,390.511,171.753,40.544,157.730
C02794=1043.485,275.907,390.543,171.750,40.542,157.729
C02795=1043.479,275.659,390.573,171.747,40.540,157.729
C02796=1043.472,275.411,390.605,171.743,40.537,157.728
C02797=1043.465,275.163,390.635,171.740,40.535,157.727
C02798=1043.458,274.915,390.666,171.737,40.533,157.727
C02799=1043.453,274.667,390.697,171.734,40.531,157.726
C02800=1043.446,274.418,390.727,171.731,40.528,157.725
C02801=1043.439,274.171,390.758,171.728,40.526,157.725
C02802=1043.432,273.922,390.789,171.725,40.524,157.724
C02803=1043.425,273.674,390.820,171.721,40.521,157.723
C02804=1043.419,273.427,390.850,171.719,40.519,157.723
C02805=1043.413,273.178,390.881,171.715,40.517,157.722
C02806=1043.406,272.930,390.912,171.712,40.514,157.722
C02807=1043.399,272.683,390.942,171.709,40.512,157.721
C02808=1043.393,272.434,390.973,171.706,40.510,157.720
C02809=1043.386,272.186,391.004,171.703,40.508,157.720
C02810=1043.379,271.938,391.034,171.700,40.506,157.719
C02811=1043.373,271.690,391.065,171.697,40.503,157.718
C02812=1043.366,271.443,391.095,171.693,40.501,157.718
C02813=1043.359,271.194,391.126,171.691,40.499,157.717
C02814=1043.353,270.947,391.156,171.688,40.496,157.717
C02815=1043.346,270.698,391.187,171.684,40.494,157.716
C02816=1043.339,270.450,391.217,171.682,40.492,157.715
C02817=1043.332,270.202,391.248,171.678,40.490,157.715
C02818=1043.326,269.955,391.278,171.675,40.488,157.714
C02819=1043.319,269.706,391.309,171.673,40.485,157.713
C02820=1043.312,269.458,391.339,171.669,40.483,157.713
C02821=1043.306,269.210,391.369,171.666,40.481,157.712
C02822=1043.299,268.962,391.399,171.663,40.479,157.711
C02823=1043.293,268.713,391.430,171.660,40.476,157.711
C02824=1043.286,268.466,391.460,171.657,40.474,157.710
C02825=1043.280,268.217,391.490,171.654,40.472,157.710
C02826=1043.272,267.970,391.521,171.651,40.470,157.709
C02827=1043.267,267.722,391.552,171.648,40.468,157.708
C02828=1043.259,267.474,391.582,171.645,40.465,157.708
C02829=1043.254,267.226,391.612,171.642,40.463,157.707
C02830=1043.246,266.978,391.642,171.638,40.461,157.706
C02831=1043.239,266.729,391.672,171.636,40.458,157.706
C02832=1043.234,266.481,391.702,171.633,40.456,157.705
C02833=1043.227,266.233,391.732,171.629,40.454,157.705
C02834=1043.219,265.984,391.762,171.627,40.452,157.704
C02835=1043.214,265.737,391.793,171.624,40.450,157.703
C02836=1043.207,265.488,391.823,171.620,40.447,157.703
C02837=1043.200,265.241,391.852,171.618,40.445,157.702
C02838=1043.194,264.992,391.883,171.615,40.443,157.702
C02839=1043.187,264.745,391.913,171.611,40.441,157.701
C02840=1043.180,264.497,391.943,171.609,40.439,157.700
C02841=1043.173,264.248,391.974,171.606,40.437,157.700
C02842=1043.167,264.000,392.003,171.603,40.434,157.699
C02843=1043.160,263.752,392.033,171.600,40.432,157.699
C02844=1043.154,263.504,392.063,171.597,40.430,157.698
C02845=1043.146,263.215,392.098,171.593,40.427,157.697
C02846=1043.138,262.926,392.133,171.590,40.425,157.697
C02847=1043.131,262.639,392.168,171.587,40.422,157.696
C02848=1043.123,262.350,392.202,171.583,40.420,157.695
C02849=1043.117,262.102,392.233,171.581,40.417,157.695
C02850=1043.110,261.853,392.262,171.577,40.415,157.694
C02851=1043.103,261.605,392.292,171.574,40.414,157.693
C02852=1043.096,261.356,392.322,171.572,40.411,157.693
C02853=1043.090,261.109,392.351,171.569,40.409,157.692
C02854=1043.082,260.861,392.381,171.566,40.407,157.692
C02855=1043.076,260.613,392.410,171.563,40.405,157.691
C02856=1043.068,260.365,392.440,171.560,40.403,157.690
C02857=1043.062,260.116,392.469,171.557,40.401,157.690
C02858=1043.055,259.868,392.499,171.554,40.399,157.689
C02859=1043.049,259.620,392.528,171.551,40.397,157.689
C02860=1043.042,259.372,392.558,171.548,40.395,157.688
C02861=1043.035,259.124,392.587,171.545,40.392,157.688
C02862=1043.028,258.876,392.618,171.543,40.390,157.687
C02863=1043.022,258.627,392.647,171.540,40.388,157.686
C02864=1043.015,258.379,392.677,171.536,40.386,157.686
C02865=1043.009,258.131,392.706,171.534,40.384,157.685
C02866=1043.001,257.883,392.736,171.531,40.382,157.685
C02867=1042.995,257.635,392.765,171.529,40.380,157.684
C02868=1042.988,257.386,392.794,171.525,40.378,157.683
C02869=1042.982,257.138,392.824,171.522,40.375,157.683
C02870=1042.975,256.890,392.853,171.520,40.373,157.682
C02871=1042.968,256.642,392.883,171.517,40.371,157.682
C02872=1042.961,256.394,392.912,171.514,40.369,157.681
C02873=1042.955,256.145,392.941,171.511,40.367,157.681
C02874=1042.948,255.898,392.971,171.508,40.365,157.680
C02875=1042.941,255.649,393.000,171.506,40.363,157.679
C02876=1042.935,255.401,393.029,171.502,40.361,157.679
C02877=1042.928,255.153,393.059,171.499,40.358,157.678
C02878=1042.921,254.905,393.088,171.497,40.357,157.678
C02879=1042.915,254.656,393.117,171.494,40.355,157.677
C02880=1042.908,254.408,393.148,171.492,40.352,157.677
C02881=1042.902,254.160,393.177,171.488,40.350,157.676
C02882=1042.895,253.911,393.206,171.485,40.348,157.675
C02883=1042.888,253.663,393.234,171.483,40.346,157.675
C02884=1042.881,253.416,393.264,171.480,40.343,157.674
C02885=1042.875,253.167,393.294,171.478,40.342,157.674
C02886=1042.868,252.919,393.323,171.474,40.340,157.673
C02887=1042.862,252.671,393.352,171.471,40.337,157.672
C02888=1042.855,252.422,393.381,171.469,40.335,157.672
C02889=1042.849,252.174,393.411,171.466,40.333,157.671
C02890=1042.842,251.926,393.440,171.463,40.331,157.671
C02891=1042.836,251.678,393.469,171.461,40.329,157.670
C02892=1042.829,251.429,393.498,171.458,40.326,157.670
C02893=1042.822,251.182,393.527,171.455,40.325,157.669
C02894=1042.816,250.933,393.556,171.452,40.323,157.668
C02895=1042.809,250.685,393.585,171.449,40.320,157.668
C02896=1042.803,250.437,393.615,171.447,40.318,157.667
C02897=1042.796,250.189,393.644,171.444,40.316,157.667
C02898=1042.790,249.941,393.673,171.442,40.314,157.666
C02899=1042.783,249.692,393.703,171.439,40.311,157.665
C02900=1042.777,249.444,393.732,171.435,40.310,157.665
C02901=1042.770,249.154,393.765,171.433,40.307,157.664
C02902=1042.762,248.864,393.799,171.429,40.305,157.664
C02903=1042.754,248.574,393.833,171.426,40.302,157.663
C02904=1042.746,248.283,393.867,171.423,40.299,157.662
C02905=1042.740,248.035,393.896,171.420,40.298,157.662
C02906=1042.734,247.787,393.925,171.417,40.295,157.661
C02907=1042.727,247.539,393.954,171.415,40.293,157.661
C02908=1042.721,247.291,393.983,171.412,40.291,157.660
C02909=1042.714,247.042,394.012,171.409,40.289,157.659
C02910=1042.707,246.794,394.041,171.407,40.286,157.659
C02911=1042.701,246.546,394.070,171.404,40.284,157.658
C02912=1042.695,246.298,394.099,171.402,40.282,157.658
C02913=1042.689,246.050,394.128,171.399,40.280,157.657
C02914=1042.682,245.802,394.157,171.396,40.278,157.657
C02915=1042.676,245.553,394.186,171.394,40.276,157.656
C02916=1042.669,245.305,394.215,171.391,40.274,157.655
C02917=1042.663,245.056,394.243,171.389,40.271,157.655
C02918=1042.656,244.808,394.272,171.386,40.269,157.654
C02919=1042.649,244.560,394.301,171.383,40.268,157.654
C02920=1042.643,244.312,394.330,171.380,40.265,157.653
C02921=1042.636,244.063,394.358,171.377,40.263,157.652
C02922=1042.630,243.815,394.387,171.375,40.261,157.652
C02923=1042.623,243.567,394.416,171.372,40.259,157.651
C02924=1042.616,243.319,394.444,171.370,40.257,157.651
C02925=1042.610,243.070,394.473,171.367,40.255,157.650
C02926=1042.603,242.822,394.501,171.364,40.253,157.650
C02927=1042.597,242.574,394.530,171.362,40.250,157.649
C02928=1042.591,242.325,394.559,171.359,40.249,157.649
C02929=1042.584,242.077,394.587,171.357,40.246,157.648
C02930=1042.577,241.829,394.616,171.354,40.244,157.647
C02931=1042.571,241.580,394.644,171.351,40.242,157.647
C02932=1042.564,241.332,394.673,171.349,40.240,157.646
C02933=1042.557,241.084,394.701,171.346,40.238,157.646
C02934=1042.552,240.836,394.730,171.344,40.236,157.645
C02935=1042.545,240.588,394.758,171.341,40.234,157.645
C02936=1042.538,240.338,394.787,171.339,40.232,157.644
C02937=1042.531,240.091,394.815,171.336,40.230,157.644
C02938=1042.524,239.842,394.843,171.333,40.227,157.643
C02939=1042.518,239.594,394.872,171.331,40.226,157.643
C02940=1042.511,239.346,394.900,171.328,40.224,157.642
C02941=1042.504,239.098,394.928,171.326,40.221,157.641
C02942=1042.498,238.849,394.957,171.323,40.219,157.641
C02943=1042.491,238.601,394.985,171.321,40.217,157.640
C02944=1042.485,238.353,395.013,171.318,40.215,157.640
C02945=1042.479,238.105,395.042,171.315,40.213,157.639
C02946=1042.471,237.856,395.070,171.313,40.211,157.639
C02947=1042.465,237.607,395.098,171.310,40.209,157.638
C02948=1042.458,237.359,395.127,171.308,40.207,157.638
C02949=1042.452,237.110,395.154,171.305,40.205,157.637
C02950=1042.445,236.863,395.183,171.302,40.203,157.636
C02951=1042.438,236.614,395.211,171.300,40.201,157.636
C02952=1042.432,236.365,395.239,171.297,40.199,157.635
C02953=1042.425,236.118,395.267,171.295,40.197,157.635
C02954=1042.418,235.869,395.295,171.292,40.195,157.634
C02955=1042.412,235.620,395.323,171.290,40.192,157.634
C02956=1042.405,235.373,395.352,171.287,40.191,157.633
C02957=1042.398,235.077,395.384,171.283,40.188,157.632
C02958=1042.390,234.781,395.418,171.281,40.186,157.632
C02959=1042.381,234.485,395.452,171.278,40.183,157.631
C02960=1042.374,234.189,395.485,171.274,40.181,157.631
C02961=1042.367,233.941,395.513,171.273,40.178,157.630
C02962=1042.361,233.693,395.541,171.270,40.177,157.630
C02963=1042.355,233.444,395.570,171.268,40.174,157.629
C02964=1042.348,233.195,395.597,171.265,40.172,157.628
C02965=1042.341,232.948,395.626,171.263,40.170,157.628
C02966=1042.334,232.699,395.653,171.260,40.168,157.627
C02967=1042.328,232.450,395.682,171.257,40.166,157.627
C02968=1042.322,232.202,395.709,171.255,40.164,157.626
C02969=1042.315,231.954,395.737,171.252,40.162,157.626
C02970=1042.308,231.705,395.765,171.250,40.160,157.625
C02971=1042.301,231.457,395.793,171.247,40.158,157.625
C02972=1042.295,231.209,395.821,171.245,40.156,157.624
C02973=1042.289,230.961,395.849,171.242,40.154,157.624
C02974=1042.283,230.712,395.877,171.240,40.151,157.623
C02975=1042.276,230.464,395.905,171.238,40.150,157.622
C02976=1042.269,230.215,395.932,171.235,40.147,157.622
C02977=1042.263,229.967,395.960,171.233,40.145,157.621
C02978=1042.256,229.719,395.988,171.230,40.143,157.621
C02979=1042.249,229.470,396.015,171.228,40.141,157.620
C02980=1042.243,229.222,396.043,171.225,40.139,157.620
C02981=1042.236,228.973,396.071,171.223,40.137,157.619
C02982=1042.230,228.724,396.099,171.220,40.135,157.619
C02983=1042.223,228.476,396.127,171.218,40.133,157.618
C02984=1042.217,228.229,396.154,171.216,40.131,157.618
C02985=1042.210,227.980,396.181,171.213,40.129,157.617
C02986=1042.203,227.732,396.209,171.211,40.126,157.616
C02987=1042.196,227.483,396.237,171.208,40.125,157.616
C02988=1042.190,227.235,396.265,171.206,40.123,157.615
C02989=1042.183,226.986,396.292,171.203,40.121,157.615
C02990=1042.177,226.737,396.319,171.200,40.119,157.614
C02991=1042.170,226.489,396.347,171.198,40.116,157.614
C02992=1042.163,226.240,396.375,171.196,40.115,157.613
C02993=1042.156,225.992,396.402,171.194,40.112,157.613
C02994=1042.150,225.745,396.429,171.191,40.111,157.612
C02995=1042.143,225.496,396.457,171.189,40.108,157.612
C02996=1042.137,225.247,396.484,171.186,40.106,157.611
C02997=1042.130,224.999,396.512,171.184,40.105,157.611
C02998=1042.123,224.750,396.540,171.182,40.102,157.610
C02999=1042.117,224.502,396.567,171.180,40.101,157.610
C03000=1042.111,224.254,396.595,171.177,40.098,157.609
C03001=1042.104,224.005,396.621,171.174,40.096,157.609
C03002=1042.097,223.757,396.649,171.172,40.094,157.608
C03003=1042.090,223.508,396.677,171.169,40.092,157.608
C03004=1042.084,223.260,396.704,171.168,40.090,157.607
C03005=1042.077,223.011,396.731,171.165,40.088,157.607
C03006=1042.071,222.763,396.759,171.163,40.086,157.606
C03007=1042.064,222.515,396.786,171.160,40.084,157.605
C03008=1042.057,222.266,396.813,171.158,40.082,157.605
C03009=1042.051,222.018,396.841,171.155,40.080,157.604
C03010=1042.045,221.770,396.868,171.153,40.077,157.604
C03011=1042.038,221.521,396.895,171.151,40.076,157.603
C03012=1042.031,221.272,396.923,171.148,40.073,157.603
C03013=1042.023,220.969,396.956,171.146,40.071,157.602
C03014=1042.015,220.666,396.989,171.143,40.068,157.601
C03015=1042.007,220.362,397.023,171.140,40.066,157.601
C03016=1041.999,220.060,397.055,171.137,40.063,157.600
C03017=1041.993,219.811,397.082,171.135,40.061,157.600
C03018=1041.986,219.562,397.110,171.133,40.059,157.599
C03019=1041.979,219.313,397.137,171.130,40.057,157.599
C03020=1041.973,219.066,397.164,171.128,40.055,157.598
C03021=1041.966,218.817,397.190,171.125,40.053,157.598
C03022=1041.959,218.569,397.218,171.123,40.051,157.597
C03023=1041.953,218.319,397.245,171.121,40.049,157.596
C03024=1041.946,218.072,397.272,171.118,40.047,157.596
C03025=1041.940,217.823,397.299,171.116,40.045,157.595
C03026=1041.932,217.575,397.326,171.114,40.043,157.595
C03027=1041.926,217.326,397.353,171.112,40.041,157.594
C03028=1041.919,217.078,397.380,171.109,40.039,157.594
C03029=1041.913,216.829,397.407,171.107,40.037,157.593
C03030=1041.906,216.580,397.434,171.105,40.035,157.593
C03031=1041.899,216.332,397.461,171.103,40.032,157.592
C03032=1041.893,216.084,397.488,171.100,40.031,157.592
C03033=1041.886,215.836,397.515,171.097,40.028,157.591
C03034=1041.879,215.587,397.542,171.096,40.027,157.591
C03035=1041.873,215.339,397.568,171.093,40.024,157.590
C03036=1041.866,215.090,397.595,171.091,40.022,157.590
C03037=1041.860,214.841,397.623,171.088,40.020,157.589
C03038=1041.853,214.593,397.649,171.087,40.018,157.589
C03039=1041.847,214.345,397.676,171.084,40.016,157.588
C03040=1041.839,214.096,397.703,171.082,40.014,157.588
C03041=1041.834,213.847,397.729,171.080,40.012,157.587
C03042=1041.826,213.599,397.756,171.078,40.010,157.587
C03043=1041.820,213.351,397.783,171.075,40.008,157.586
C03044=1041.813,213.102,397.810,171.072,40.006,157.585
C03045=1041.807,212.854,397.837,171.071,40.004,157.585
C03046=1041.801,212.605,397.864,171.068,40.002,157.584
C03047=1041.794,212.357,397.890,171.066,39.999,157.584
C03048=1041.787,212.108,397.917,171.064,39.998,157.583
C03049=1041.781,211.860,397.944,171.062,39.995,157.583
C03050=1041.774,211.611,397.971,171.059,39.993,157.582
C03051=1041.768,211.363,397.997,171.058,39.991,157.582
C03052=1041.761,211.114,398.024,171.055,39.989,157.581
C03053=1041.754,210.865,398.051,171.053,39.987,157.581
C03054=1041.748,210.617,398.077,171.051,39.985,157.580
C03055=1041.741,210.369,398.104,171.049,39.983,157.580
C03056=1041.734,210.121,398.130,171.046,39.981,157.579
C03057=1041.727,209.872,398.157,171.044,39.979,157.579
C03058=1041.721,209.623,398.184,171.042,39.976,157.578
C03059=1041.714,209.375,398.210,171.039,39.975,157.578
C03060=1041.707,209.126,398.236,171.038,39.972,157.577
C03061=1041.702,208.878,398.263,171.035,39.971,157.577
C03062=1041.694,208.629,398.289,171.033,39.968,157.576
C03063=1041.688,208.381,398.316,171.031,39.966,157.576
C03064=1041.682,208.132,398.343,171.029,39.964,157.575
C03065=1041.674,207.883,398.369,171.026,39.962,157.575
C03066=1041.668,207.635,398.395,171.025,39.960,157.574
C03067=1041.661,207.386,398.421,171.022,39.958,157.574
C03068=1041.655,207.138,398.448,171.020,39.956,157.573
C03069=1041.647,206.841,398.480,171.017,39.953,157.572
C03070=1041.639,206.542,398.512,171.015,39.951,157.572
C03071=1041.630,206.245,398.543,171.013,39.948,157.571
C03072=1041.622,205.947,398.574,171.010,39.946,157.571
C03073=1041.597,204.896,398.681,170.730,39.843,157.539
C03074=1041.590,204.648,398.706,170.728,39.842,157.538
C03075=1041.584,204.398,398.731,170.724,39.840,157.538
C03076=1041.578,204.150,398.756,170.721,39.839,157.537
C03077=1041.572,203.901,398.782,170.719,39.838,157.537
C03078=1041.566,203.652,398.807,170.715,39.837,157.537
C03079=1041.560,203.404,398.832,170.713,39.835,157.536
C03080=1041.553,203.155,398.858,170.710,39.834,157.536
C03081=1041.547,202.907,398.881,170.706,39.832,157.535
C03082=1041.541,202.658,398.907,170.704,39.831,157.535
C03083=1041.535,202.409,398.932,170.700,39.830,157.535
C03084=1041.529,202.161,398.957,170.698,39.829,157.534
C03085=1041.523,201.911,398.982,170.695,39.827,157.534
C03086=1041.517,201.663,399.007,170.692,39.826,157.534
C03087=1041.511,201.415,399.032,170.689,39.824,157.533
C03088=1041.505,201.166,399.058,170.686,39.823,157.533
C03089=1041.499,200.917,399.082,170.683,39.822,157.533
C03090=1041.492,200.668,399.107,170.680,39.821,157.532
C03091=1041.486,200.419,399.132,170.678,39.820,157.532
C03092=1041.479,200.171,399.156,170.674,39.819,157.531
C03093=1041.473,199.922,399.182,170.672,39.818,157.531
C03094=1041.468,199.674,399.206,170.668,39.816,157.531
C03095=1041.461,199.425,399.231,170.665,39.815,157.530
C03096=1041.455,199.176,399.255,170.663,39.814,157.530
C03097=1041.448,198.927,399.280,170.660,39.813,157.530
C03098=1041.442,198.678,399.305,170.657,39.811,157.529
C03099=1041.436,198.431,399.329,170.654,39.810,157.529
C03100=1041.430,198.181,399.354,170.652,39.809,157.529
C03101=1041.423,197.933,399.379,170.648,39.808,157.528
C03102=1041.417,197.684,399.403,170.645,39.807,157.528
C03103=1041.411,197.435,399.428,170.642,39.806,157.528
C03104=1041.405,197.187,399.452,170.639,39.805,157.527
C03105=1041.398,196.938,399.477,170.637,39.804,157.527
C03106=1041.392,196.689,399.501,170.633,39.802,157.527
C03107=1041.386,196.440,399.527,170.631,39.801,157.526
C03108=1041.380,196.192,399.551,170.628,39.800,157.526
C03109=1041.374,195.943,399.575,170.626,39.799,157.526
C03110=1041.367,195.694,399.600,170.622,39.798,157.525
C03111=1041.361,195.445,399.624,170.620,39.796,157.525
C03112=1041.355,195.197,399.649,170.617,39.795,157.525
C03113=1041.349,194.948,399.673,170.614,39.794,157.524
C03114=1041.343,194.699,399.698,170.611,39.793,157.524
C03115=1041.336,194.451,399.722,170.609,39.792,157.524
C03116=1041.330,194.202,399.747,170.605,39.791,157.523
C03117=1041.324,193.953,399.772,170.603,39.789,157.523
C03118=1041.318,193.705,399.796,170.600,39.788,157.523
C03119=1041.312,193.456,399.821,170.597,39.787,157.522
C03120=1041.306,193.207,399.845,170.594,39.786,157.522
C03121=1041.300,192.959,399.870,170.592,39.785,157.521
C03122=1041.293,192.710,399.894,170.588,39.784,157.521
C03123=1041.287,192.461,399.918,170.586,39.783,157.521
C03124=1041.281,192.212,399.942,170.583,39.782,157.521
C03125=1041.275,191.964,399.967,170.580,39.781,157.520
C03126=1041.269,191.715,399.991,170.577,39.780,157.520
C03127=1041.263,191.466,400.015,170.575,39.779,157.520
C03128=1041.257,191.217,400.040,170.571,39.777,157.519
C03129=1041.251,190.968,400.064,170.569,39.776,157.519
C03130=1041.244,190.720,400.089,170.566,39.775,157.519
C03131=1041.238,190.471,400.113,170.563,39.774,157.518
C03132=1041.232,190.223,400.137,170.561,39.773,157.518
C03133=1041.227,189.973,400.161,170.558,39.772,157.518
C03134=1041.219,189.689,400.189,170.554,39.770,157.517
C03135=1041.213,189.405,400.216,170.551,39.769,157.517
C03136=1041.205,189.121,400.245,170.549,39.767,157.516
C03137=1041.199,188.835,400.272,170.545,39.766,157.516
C03138=1041.193,188.587,400.296,170.543,39.765,157.516
C03139=1041.187,188.338,400.321,170.540,39.764,157.515
C03140=1041.181,188.090,400.344,170.537,39.763,157.515
C03141=1041.175,187.840,400.369,170.534,39.762,157.515
C03142=1041.169,187.593,400.393,170.532,39.761,157.514
C03143=1041.163,187.343,400.418,170.528,39.760,157.514
C03144=1041.157,187.095,400.442,170.526,39.759,157.514
C03145=1041.151,186.846,400.466,170.524,39.758,157.513
C03146=1041.145,186.598,400.490,170.521,39.757,157.513
C03147=1041.139,186.348,400.515,170.518,39.755,157.513
C03148=1041.133,186.100,400.538,170.515,39.754,157.513
C03149=1041.127,185.851,400.563,170.513,39.753,157.512
C03150=1041.121,185.602,400.587,170.510,39.752,157.512
C03151=1041.114,185.353,400.611,170.507,39.751,157.512
C03152=1041.109,185.105,400.635,170.505,39.750,157.511
C03153=1041.103,184.856,400.659,170.501,39.749,157.511
C03154=1041.098,184.607,400.682,170.499,39.748,157.511
C03155=1041.091,184.358,400.706,170.497,39.746,157.510
C03156=1041.086,184.109,400.731,170.493,39.746,157.510
C03157=1041.080,183.861,400.754,170.491,39.744,157.510
C03158=1041.074,183.612,400.779,170.489,39.743,157.509
C03159=1041.068,183.363,400.803,170.486,39.742,157.509
C03160=1041.061,183.114,400.827,170.483,39.741,157.509
C03161=1041.055,182.865,400.850,170.480,39.741,157.509
C03162=1041.049,182.616,400.874,170.478,39.740,157.508
C03163=1041.042,182.368,400.897,170.474,39.739,157.508
C03164=1041.036,182.119,400.920,170.472,39.738,157.508
C03165=1041.029,181.871,400.944,170.470,39.737,157.507
C03166=1041.023,181.622,400.968,170.467,39.736,157.507
C03167=1041.017,181.373,400.991,170.464,39.735,157.507
C03168=1041.010,181.124,401.015,170.461,39.734,157.506
C03169=1041.004,180.875,401.038,170.459,39.734,157.506
C03170=1040.998,180.626,401.062,170.457,39.733,157.506
C03171=1040.992,180.378,401.085,170.453,39.732,157.506
C03172=1040.985,180.129,401.109,170.451,39.731,157.505
C03173=1040.980,179.880,401.132,170.448,39.730,157.505
C03174=1040.973,179.631,401.156,170.446,39.729,157.505
C03175=1040.967,179.382,401.179,170.443,39.728,157.505
C03176=1040.960,179.133,401.203,170.440,39.727,157.504
C03177=1040.954,178.885,401.226,170.438,39.727,157.504
C03178=1040.948,178.635,401.250,170.435,39.726,157.504
C03179=1040.942,178.387,401.273,170.432,39.725,157.503
C03180=1040.936,178.138,401.296,170.430,39.724,157.503
C03181=1040.929,177.889,401.320,170.427,39.723,157.503
C03182=1040.923,177.640,401.343,170.425,39.722,157.503
C03183=1040.917,177.391,401.367,170.422,39.721,157.502
C03184=1040.911,177.142,401.390,170.419,39.721,157.502
C03185=1040.904,176.894,401.413,170.417,39.720,157.502
C03186=1040.898,176.645,401.437,170.415,39.718,157.502
C03187=1040.892,176.397,401.460,170.411,39.717,157.501
C03188=1040.886,176.148,401.483,170.409,39.717,157.501
C03189=1040.880,175.899,401.507,170.406,39.716,157.501
C03190=1040.874,175.650,401.530,170.403,39.715,157.500
C03191=1040.867,175.401,401.554,170.401,39.715,157.500
C03192=1040.861,175.152,401.577,170.398,39.714,157.500
C03193=1040.855,174.903,401.600,170.396,39.712,157.500
C03194=1040.848,174.654,401.624,170.393,39.711,157.499
C03195=1040.843,174.405,401.646,170.390,39.711,157.499
C03196=1040.837,174.157,401.670,170.388,39.710,157.499
C03197=1040.830,173.908,401.693,170.386,39.709,157.499
C03198=1040.823,173.623,401.719,170.382,39.708,157.498
C03199=1040.816,173.338,401.747,170.380,39.707,157.498
C03200=1040.810,173.053,401.773,170.377,39.706,157.498
C03201=1040.802,172.769,401.800,170.374,39.705,157.497
C03202=1040.797,172.520,401.822,170.371,39.704,157.497
C03203=1040.790,172.270,401.846,170.369,39.703,157.497
C03204=1040.784,172.022,401.869,170.366,39.702,157.497
C03205=1040.779,171.773,401.892,170.364,39.702,157.496
C03206=1040.772,171.525,401.915,170.361,39.701,157.496
C03207=1040.765,171.276,401.939,170.358,39.700,157.496
C03208=1040.760,171.027,401.962,170.356,39.699,157.496
C03209=1040.754,170.778,401.985,170.354,39.698,157.495
C03210=1040.748,170.529,402.008,170.351,39.697,157.495
C03211=1040.742,170.280,402.032,170.348,39.697,157.495
C03212=1040.735,170.031,402.054,170.346,39.696,157.495
C03213=1040.729,169.783,402.077,170.344,39.694,157.494
C03214=1040.724,169.534,402.100,170.340,39.694,157.494
C03215=1040.717,169.284,402.123,170.338,39.693,157.494
C03216=1040.711,169.036,402.147,170.336,39.692,157.493
C03217=1040.706,168.787,402.170,170.334,39.691,157.493
C03218=1040.699,168.538,402.192,170.330,39.690,157.493
C03219=1040.693,168.289,402.215,170.328,39.689,157.493
C03220=1040.688,168.040,402.238,170.326,39.689,157.492
C03221=1040.681,167.791,402.261,170.324,39.688,157.492
C03222=1040.675,167.543,402.285,170.320,39.687,157.492
C03223=1040.669,167.294,402.307,170.318,39.686,157.492
C03224=1040.663,167.045,402.330,170.316,39.685,157.491
C03225=1040.657,166.796,402.353,170.314,39.684,157.491
C03226=1040.652,166.547,402.376,170.310,39.684,157.491
C03227=1040.646,166.298,402.399,170.308,39.683,157.491
C03228=1040.640,166.049,402.422,170.306,39.682,157.490
C03229=1040.633,165.800,402.445,170.304,39.681,157.490
C03230=1040.627,165.551,402.468,170.301,39.680,157.490
C03231=1040.622,165.302,402.491,170.298,39.679,157.490
C03232=1040.616,165.054,402.514,170.296,39.679,157.489
C03233=1040.610,164.805,402.537,170.294,39.678,157.489
C03234=1040.603,164.557,402.560,170.291,39.677,157.489
C03235=1040.598,164.308,402.583,170.288,39.676,157.489
C03236=1040.592,164.059,402.606,170.286,39.675,157.488
C03237=1040.586,163.810,402.629,170.284,39.674,157.488
C03238=1040.580,163.560,402.652,170.281,39.673,157.488
C03239=1040.573,163.312,402.674,170.279,39.672,157.487
C03240=1040.568,163.063,402.697,170.276,39.671,157.487
C03241=1040.562,162.814,402.720,170.274,39.671,157.487
C03242=1040.556,162.565,402.743,170.271,39.670,157.487
C03243=1040.550,162.316,402.765,170.269,39.669,157.486
C03244=1040.544,162.067,402.788,170.267,39.668,157.486
C03245=1040.539,161.818,402.811,170.265,39.667,157.486
C03246=1040.533,161.569,402.833,170.261,39.666,157.486
C03247=1040.527,161.320,402.856,170.259,39.666,157.485
C03248=1040.521,161.072,402.879,170.257,39.665,157.485
C03249=1040.515,160.823,402.902,170.255,39.664,157.485
C03250=1040.509,160.574,402.925,170.253,39.663,157.485
C03251=1040.503,160.325,402.948,170.249,39.662,157.484
C03252=1040.497,160.076,402.969,170.247,39.662,157.484
C03253=1040.492,159.827,402.992,170.245,39.661,157.484
C03254=1040.485,159.578,403.015,170.243,39.660,157.484
C03255=1040.479,159.330,403.037,170.240,39.659,157.483
C03256=1040.473,159.080,403.059,170.237,39.659,157.483
C03257=1040.467,158.832,403.081,170.235,39.658,157.483
C03258=1040.461,158.583,403.104,170.233,39.657,157.483
C03259=1040.455,158.334,403.127,170.231,39.657,157.483
C03260=1040.448,158.084,403.149,170.228,39.656,157.482
C03261=1040.442,157.835,403.172,170.225,39.655,157.482
C03262=1040.435,157.550,403.197,170.223,39.654,157.482
C03263=1040.428,157.265,403.223,170.220,39.654,157.482
C03264=1040.421,156.980,403.248,170.217,39.653,157.481
C03265=1040.414,156.695,403.274,170.214,39.652,157.481
C03266=1040.408,156.445,403.296,170.212,39.651,157.481
C03267=1040.402,156.197,403.318,170.210,39.650,157.481
C03268=1040.396,155.948,403.341,170.208,39.650,157.480
C03269=1040.390,155.699,403.363,170.205,39.649,157.480
C03270=1040.384,155.450,403.385,170.202,39.648,157.480
C03271=1040.377,155.202,403.408,170.200,39.648,157.480
C03272=1040.372,154.952,403.430,170.198,39.647,157.479
C03273=1040.365,154.703,403.452,170.195,39.646,157.479
C03274=1040.359,154.454,403.474,170.193,39.645,157.479
C03275=1040.353,154.205,403.497,170.191,39.645,157.479
C03276=1040.347,153.956,403.518,170.188,39.644,157.479
C03277=1040.341,153.708,403.541,170.186,39.643,157.478
C03278=1040.335,153.458,403.562,170.183,39.643,157.478
C03279=1040.328,153.210,403.585,170.181,39.642,157.478
C03280=1040.323,152.960,403.607,170.179,39.641,157.478
C03281=1040.316,152.712,403.629,170.177,39.641,157.478
C03282=1040.310,152.462,403.651,170.174,39.640,157.477
C03283=1040.304,152.214,403.673,170.171,39.639,157.477
C03284=1040.298,151.964,403.696,170.169,39.639,157.477
C03285=1040.292,151.716,403.718,170.167,39.638,157.477
C03286=1040.286,151.467,403.739,170.165,39.637,157.476
C03287=1040.280,151.218,403.761,170.163,39.637,157.476
C03288=1040.274,150.969,403.783,170.160,39.636,157.476
C03289=1040.268,150.720,403.805,170.157,39.635,157.476
C03290=1040.262,150.471,403.828,170.155,39.635,157.476
C03291=1040.255,150.222,403.849,170.153,39.634,157.475
C03292=1040.249,149.973,403.871,170.151,39.633,157.475
C03293=1040.243,149.724,403.893,170.148,39.633,157.475
C03294=1040.237,149.475,403.915,170.146,39.632,157.475
C03295=1040.231,149.226,403.937,170.144,39.631,157.474
C03296=1040.225,148.978,403.959,170.141,39.631,157.474
C03297=1040.219,148.729,403.981,170.139,39.630,157.474
C03298=1040.213,148.479,404.002,170.136,39.629,157.474
C03299=1040.207,148.231,404.025,170.134,39.629,157.474
C03300=1040.200,147.982,404.046,170.132,39.628,157.474
C03301=1040.194,147.732,404.068,170.130,39.627,157.473
C03302=1040.188,147.484,404.090,170.128,39.627,157.473
C03303=1040.182,147.234,404.113,170.126,39.626,157.473
C03304=1040.177,146.986,404.134,170.122,39.625,157.473
C03305=1040.171,146.737,404.156,170.120,39.625,157.472
C03306=1040.164,146.487,404.177,170.118,39.624,157.472
C03307=1040.158,146.239,404.200,170.116,39.624,157.472
C03308=1040.152,145.990,404.221,170.114,39.623,157.472
C03309=1040.145,145.741,404.242,170.111,39.622,157.472
C03310=1040.139,145.491,404.264,170.109,39.622,157.471
C03311=1040.133,145.243,404.285,170.107,39.621,157.471
C03312=1040.127,144.994,404.308,170.104,39.621,157.471
C03313=1040.121,144.745,404.329,170.102,39.620,157.471
C03314=1040.114,144.496,404.351,170.099,39.619,157.471
C03315=1040.108,144.247,404.372,170.097,39.619,157.470
C03316=1040.102,143.998,404.394,170.095,39.618,157.470
C03317=1040.097,143.749,404.415,170.093,39.617,157.470
C03318=1040.090,143.500,404.437,170.091,39.617,157.470
C03319=1040.084,143.251,404.459,170.089,39.616,157.470
C03320=1040.078,143.001,404.480,170.086,39.616,157.469
C03321=1040.072,142.753,404.503,170.083,39.616,157.469
C03322=1040.066,142.504,404.524,170.081,39.614,157.469
C03323=1040.060,142.255,404.545,170.079,39.614,157.469
C03324=1040.054,142.006,404.567,170.077,39.614,157.469
C03325=1040.047,141.757,404.588,170.074,39.613,157.468
C03326=1040.041,141.471,404.612,170.072,39.612,157.468
C03327=1040.033,141.186,404.638,170.069,39.612,157.468
C03328=1040.027,140.900,404.663,170.067,39.610,157.468
C03329=1040.019,140.614,404.687,170.065,39.610,157.468
C03330=1040.013,140.365,404.708,170.061,39.610,157.467
C03331=1040.007,140.117,404.730,170.059,39.609,157.467
C03332=1040.001,139.867,404.751,170.057,39.608,157.467
C03333=1039.995,139.618,404.773,170.055,39.608,157.467
C03334=1039.989,139.369,404.795,170.053,39.607,157.467
C03335=1039.983,139.120,404.816,170.051,39.607,157.466
C03336=1039.976,138.872,404.837,170.048,39.606,157.466
C03337=1039.970,138.622,404.858,170.046,39.605,157.466
C03338=1039.964,138.373,404.880,170.044,39.605,157.466
C03339=1039.959,138.125,404.901,170.042,39.604,157.466
C03340=1039.952,137.875,404.922,170.040,39.604,157.465
C03341=1039.946,137.626,404.943,170.038,39.603,157.465
C03342=1039.940,137.377,404.965,170.034,39.603,157.465
C03343=1039.934,137.128,404.986,170.032,39.602,157.465
C03344=1039.927,136.879,405.007,170.030,39.601,157.465
C03345=1039.921,136.630,405.029,170.028,39.601,157.464
C03346=1039.915,136.382,405.050,170.026,39.600,157.464
C03347=1039.909,136.132,405.071,170.023,39.600,157.464
C03348=1039.903,135.883,405.092,170.021,39.599,157.464
C03349=1039.897,135.634,405.113,170.019,39.599,157.464
C03350=1039.890,135.386,405.134,170.017,39.598,157.464
C03351=1039.884,135.136,405.156,170.015,39.598,157.463
C03352=1039.878,134.886,405.177,170.013,39.597,157.463
C03353=1039.872,134.638,405.198,170.010,39.596,157.463
C03354=1039.866,134.389,405.219,170.008,39.596,157.463
C03355=1039.860,134.140,405.241,170.006,39.595,157.463
C03356=1039.854,133.891,405.261,170.004,39.595,157.462
C03357=1039.847,133.642,405.283,170.002,39.595,157.462
C03358=1039.841,133.393,405.304,169.999,39.594,157.462
C03359=1039.835,133.144,405.324,169.997,39.594,157.462
C03360=1039.829,132.895,405.346,169.994,39.593,157.462
C03361=1039.824,132.646,405.367,169.992,39.592,157.461
C03362=1039.817,132.397,405.387,169.990,39.592,157.461
C03363=1039.811,132.147,405.409,169.988,39.591,157.461
C03364=1039.805,131.899,405.430,169.986,39.591,157.461
C03365=1039.798,131.650,405.451,169.983,39.590,157.461
C03366=1039.793,131.400,405.472,169.981,39.590,157.461
C03367=1039.787,131.152,405.494,169.979,39.589,157.460
C03368=1039.780,130.902,405.514,169.977,39.588,157.460
C03369=1039.773,130.653,405.535,169.975,39.588,157.460
C03370=1039.768,130.404,405.555,169.973,39.587,157.460
C03371=1039.761,130.155,405.576,169.971,39.587,157.460
C03372=1039.755,129.906,405.598,169.968,39.587,157.460
C03373=1039.749,129.657,405.618,169.966,39.586,157.459
C03374=1039.742,129.408,405.639,169.964,39.586,157.459
C03375=1039.736,129.159,405.660,169.962,39.586,157.459
C03376=1039.730,128.910,405.681,169.960,39.585,157.459
C03377=1039.723,128.661,405.701,169.957,39.585,157.459
C03378=1039.718,128.412,405.722,169.955,39.584,157.459
C03379=1039.711,128.163,405.743,169.952,39.584,157.458
C03380=1039.705,127.913,405.763,169.950,39.583,157.458
C03381=1039.699,127.665,405.784,169.948,39.583,157.458
C03382=1039.693,127.415,405.805,169.946,39.582,157.458
C03383=1039.686,127.167,405.825,169.944,39.582,157.458
C03384=1039.680,126.917,405.846,169.942,39.581,157.458
C03385=1039.674,126.668,405.867,169.939,39.581,157.457
C03386=1039.668,126.420,405.887,169.937,39.580,157.457
C03387=1039.661,126.170,405.909,169.935,39.580,157.457
C03388=1039.655,125.922,405.929,169.933,39.579,157.457
C03389=1039.649,125.672,405.949,169.931,39.579,157.457
C03390=1039.642,125.387,405.973,169.929,39.579,157.457
C03391=1039.634,125.101,405.997,169.926,39.578,157.456
C03392=1039.627,124.815,406.020,169.923,39.578,157.456
C03393=1039.621,124.529,406.044,169.921,39.577,157.456
C03394=1039.614,124.280,406.065,169.919,39.576,157.456
C03395=1039.608,124.030,406.085,169.917,39.576,157.456
C03396=1039.602,123.782,406.105,169.915,39.575,157.455
C03397=1039.596,123.532,406.127,169.913,39.575,157.455
C03398=1039.590,123.284,406.147,169.910,39.574,157.455
C03399=1039.583,123.034,406.167,169.908,39.574,157.455
C03400=1039.577,122.786,406.188,169.906,39.573,157.455
C03401=1039.571,122.536,406.209,169.904,39.573,157.455
C03402=1039.565,122.287,406.229,169.902,39.572,157.454
C03403=1039.559,122.038,406.250,169.899,39.572,157.454
C03404=1039.553,121.789,406.270,169.896,39.571,157.454
C03405=1039.546,121.540,406.291,169.894,39.571,157.454
C03406=1039.541,121.291,406.311,169.892,39.571,157.454
C03407=1039.534,121.042,406.332,169.890,39.570,157.454
C03408=1039.528,120.793,406.352,169.888,39.570,157.453
C03409=1039.521,120.543,406.373,169.887,39.569,157.453
C03410=1039.516,120.294,406.393,169.885,39.569,157.453
C03411=1039.510,120.046,406.414,169.882,39.568,157.453
C03412=1039.503,119.796,406.434,169.880,39.568,157.453
C03413=1039.498,119.547,406.455,169.878,39.567,157.453
C03414=1039.491,119.298,406.475,169.876,39.567,157.452
C03415=1039.485,119.049,406.495,169.874,39.566,157.452
C03416=1039.478,118.800,406.516,169.872,39.566,157.452
C03417=1039.473,118.551,406.537,169.870,39.565,157.452
C03418=1039.467,118.302,406.557,169.867,39.565,157.452
C03419=1039.461,118.053,406.577,169.865,39.564,157.452
C03420=1039.455,117.804,406.597,169.863,39.564,157.451
C03421=1039.449,117.554,406.618,169.861,39.563,157.451
C03422=1039.442,117.306,406.638,169.859,39.563,157.451
C03423=1039.436,117.056,406.659,169.857,39.562,157.451
C03424=1039.431,116.807,406.679,169.854,39.562,157.451
C03425=1039.425,116.558,406.699,169.852,39.561,157.451
C03426=1039.418,116.309,406.720,169.850,39.561,157.451
C03427=1039.412,116.060,406.739,169.848,39.561,157.450
C03428=1039.407,115.811,406.760,169.846,39.560,157.450
C03429=1039.400,115.561,406.780,169.844,39.560,157.450
C03430=1039.394,115.313,406.800,169.842,39.559,157.450
C03431=1039.388,115.063,406.821,169.839,39.559,157.450
C03432=1039.382,114.815,406.842,169.837,39.558,157.450
C03433=1039.376,114.566,406.862,169.835,39.558,157.449
C03434=1039.369,114.316,406.882,169.833,39.557,157.449
C03435=1039.364,114.067,406.903,169.831,39.557,157.449
C03436=1039.358,113.818,406.923,169.829,39.556,157.449
C03437=1039.352,113.569,406.943,169.826,39.555,157.449
C03438=1039.346,113.320,406.963,169.824,39.555,157.449
C03439=1039.340,113.071,406.983,169.822,39.555,157.448
C03440=1039.333,112.822,407.003,169.820,39.554,157.448
C03441=1039.327,112.573,407.023,169.819,39.554,157.448
C03442=1039.321,112.323,407.042,169.817,39.553,157.448
C03443=1039.315,112.074,407.063,169.815,39.553,157.448
C03444=1039.309,111.825,407.083,169.812,39.552,157.448
C03445=1039.302,111.576,407.103,169.810,39.552,157.447
C03446=1039.296,111.327,407.123,169.808,39.551,157.447
C03447=1039.290,111.078,407.143,169.806,39.551,157.447
C03448=1039.284,110.828,407.163,169.804,39.550,157.447
C03449=1039.278,110.580,407.183,169.802,39.550,157.447
C03450=1039.272,110.331,407.203,169.800,39.550,157.447
C03451=1039.265,110.081,407.223,169.798,39.550,157.446
C03452=1039.259,109.832,407.243,169.795,39.549,157.446
C03453=1039.253,109.583,407.263,169.793,39.549,157.446
C03454=1039.246,109.297,407.285,169.791,39.548,157.446
C03455=1039.238,109.011,407.308,169.788,39.548,157.446
C03456=1039.231,108.725,407.331,169.786,39.547,157.446
C03457=1039.224,108.439,407.354,169.784,39.547,157.445
C03458=1039.218,108.190,407.373,169.782,39.546,157.445
C03459=1039.211,107.941,407.393,169.779,39.547,157.445
C03460=1039.205,107.691,407.413,169.777,39.546,157.445
C03461=1039.199,107.443,407.433,169.775,39.546,157.445
C03462=1039.193,107.193,407.453,169.773,39.545,157.445
C03463=1039.187,106.944,407.473,169.771,39.545,157.445
C03464=1039.180,106.695,407.492,169.769,39.544,157.444
C03465=1039.174,106.446,407.511,169.767,39.544,157.444
C03466=1039.168,106.197,407.532,169.765,39.544,157.444
C03467=1039.162,105.947,407.551,169.762,39.543,157.444
C03468=1039.156,105.699,407.571,169.760,39.543,157.444
C03469=1039.149,105.449,407.591,169.758,39.542,157.444
C03470=1039.143,105.201,407.611,169.756,39.542,157.444
C03471=1039.137,104.951,407.630,169.754,39.542,157.443
C03472=1039.131,104.702,407.650,169.752,39.541,157.443
C03473=1039.125,104.452,407.670,169.750,39.541,157.443
C03474=1039.119,104.203,407.689,169.748,39.541,157.443
C03475=1039.112,103.955,407.709,169.745,39.540,157.443
C03476=1039.106,103.706,407.728,169.743,39.540,157.443
C03477=1039.100,103.456,407.748,169.742,39.539,157.443
C03478=1039.094,103.207,407.768,169.740,39.539,157.442
C03479=1039.088,102.958,407.788,169.738,39.538,157.442
C03480=1039.081,102.709,407.807,169.736,39.538,157.442
C03481=1039.076,102.460,407.826,169.733,39.537,157.442
C03482=1039.069,102.210,407.847,169.731,39.537,157.442
C03483=1039.063,101.961,407.866,169.729,39.537,157.442
C03484=1039.057,101.712,407.886,169.727,39.537,157.442
C03485=1039.051,101.464,407.905,169.725,39.536,157.441
C03486=1039.045,101.214,407.924,169.723,39.536,157.441
C03487=1039.038,100.965,407.945,169.721,39.535,157.441
C03488=1039.033,100.715,407.964,169.719,39.535,157.441
C03489=1039.027,100.466,407.984,169.716,39.534,157.441
C03490=1039.020,100.217,408.003,169.714,39.534,157.441
C03491=1039.014,99.968,408.022,169.712,39.534,157.441
C03492=1039.007,99.719,408.042,169.710,39.533,157.440
C03493=1039.001,99.470,408.061,169.708,39.533,157.440
C03494=1038.995,99.221,408.080,169.707,39.532,157.440
C03495=1038.989,98.972,408.100,169.705,39.532,157.440
C03496=1038.982,98.723,408.119,169.703,39.532,157.440
C03497=1038.976,98.473,408.138,169.701,39.531,157.440
C03498=1038.970,98.224,408.158,169.698,39.531,157.440
C03499=1038.964,97.975,408.177,169.696,39.531,157.439
C03500=1038.958,97.726,408.197,169.694,39.531,157.439
C03501=1038.951,97.477,408.216,169.692,39.530,157.439
C03502=1038.945,97.227,408.235,169.690,39.530,157.439
C03503=1038.938,96.978,408.255,169.688,39.529,157.439
C03504=1038.933,96.729,408.274,169.686,39.529,157.439
C03505=1038.926,96.480,408.292,169.684,39.529,157.439
C03506=1038.920,96.231,408.312,169.681,39.528,157.438
C03507=1038.914,95.982,408.331,169.679,39.528,157.438
C03508=1038.908,95.732,408.350,169.677,39.527,157.438
C03509=1038.901,95.483,408.370,169.675,39.528,157.438
C03510=1038.895,95.234,408.389,169.673,39.527,157.438
C03511=1038.889,94.984,408.408,169.671,39.527,157.438
C03512=1038.883,94.736,408.428,169.669,39.526,157.438
C03513=1038.876,94.486,408.446,169.667,39.526,157.437
C03514=1038.870,94.237,408.466,169.666,39.526,157.437
C03515=1038.864,93.989,408.485,169.663,39.525,157.437
C03516=1038.858,93.739,408.504,169.661,39.525,157.437
C03517=1038.851,93.489,408.523,169.659,39.524,157.437
C03518=1038.845,93.204,408.546,169.657,39.524,157.437
C03519=1038.838,92.918,408.568,169.654,39.524,157.437
C03520=1038.831,92.631,408.589,169.652,39.523,157.436
C03521=1038.823,92.346,408.612,169.650,39.523,157.436
C03522=1038.817,92.096,408.630,169.647,39.523,157.436
C03523=1038.811,91.847,408.649,169.645,39.522,157.436
C03524=1038.804,91.599,408.669,169.643,39.522,157.436
C03525=1038.799,91.349,408.688,169.641,39.521,157.436
C03526=1038.792,91.100,408.707,169.639,39.521,157.436
C03527=1038.787,90.851,408.726,169.637,39.521,157.435
C03528=1038.780,90.601,408.745,169.635,39.520,157.435
C03529=1038.774,90.352,408.764,169.634,39.520,157.435
C03530=1038.768,90.104,408.783,169.631,39.519,157.435
C03531=1038.761,89.853,408.803,169.629,39.519,157.435
C03532=1038.755,89.604,408.821,169.627,39.519,157.435
C03533=1038.749,89.355,408.840,169.625,39.519,157.435
C03534=1038.742,89.106,408.859,169.623,39.518,157.434
C03535=1038.736,88.857,408.878,169.621,39.518,157.434
C03536=1038.730,88.607,408.897,169.619,39.518,157.434
C03537=1038.724,88.358,408.915,169.617,39.517,157.434
C03538=1038.717,88.109,408.934,169.615,39.518,157.434
C03539=1038.711,87.860,408.953,169.612,39.517,157.434
C03540=1038.705,87.611,408.972,169.610,39.517,157.434
C03541=1038.699,87.362,408.990,169.608,39.517,157.434
C03542=1038.692,87.112,409.009,169.606,39.516,157.434
C03543=1038.686,86.863,409.028,169.604,39.516,157.433
C03544=1038.679,86.614,409.046,169.602,39.515,157.433
C03545=1038.674,86.365,409.066,169.600,39.515,157.433
C03546=1038.667,86.116,409.084,169.598,39.515,157.433
C03547=1038.661,85.866,409.103,169.596,39.514,157.433
C03548=1038.654,85.617,409.122,169.595,39.515,157.433
C03549=1038.649,85.368,409.141,169.592,39.514,157.433
C03550=1038.642,85.119,409.159,169.590,39.514,157.432
C03551=1038.636,84.870,409.178,169.588,39.513,157.432
C03552=1038.629,84.621,409.197,169.586,39.513,157.432
C03553=1038.623,84.371,409.215,169.584,39.513,157.432
C03554=1038.617,84.122,409.235,169.582,39.512,157.432
C03555=1038.611,83.873,409.253,169.580,39.512,157.432
C03556=1038.604,83.624,409.272,169.578,39.512,157.432
C03557=1038.598,83.375,409.291,169.575,39.511,157.432
C03558=1038.592,83.125,409.309,169.573,39.511,157.431
C03559=1038.585,82.876,409.327,169.571,39.511,157.431
C03560=1038.580,82.626,409.346,169.569,39.511,157.431
C03561=1038.573,82.377,409.365,169.567,39.510,157.431
C03562=1038.567,82.128,409.384,169.565,39.510,157.431
C03563=1038.561,81.879,409.402,169.564,39.510,157.431
C03564=1038.554,81.630,409.421,169.562,39.509,157.431
C03565=1038.549,81.380,409.440,169.560,39.509,157.431
C03566=1038.542,81.131,409.458,169.557,39.508,157.430
C03567=1038.536,80.882,409.477,169.555,39.509,157.430
C03568=1038.529,80.632,409.496,169.553,39.508,157.430
C03569=1038.523,80.383,409.514,169.551,39.508,157.430
C03570=1038.517,80.134,409.533,169.549,39.507,157.430
C03571=1038.511,79.884,409.551,169.547,39.507,157.430
C03572=1038.505,79.636,409.570,169.545,39.507,157.430
C03573=1038.499,79.387,409.588,169.543,39.506,157.429
C03574=1038.493,79.137,409.607,169.540,39.506,157.429
C03575=1038.486,78.888,409.626,169.539,39.506,157.429
C03576=1038.480,78.639,409.644,169.537,39.505,157.429
C03577=1038.474,78.389,409.663,169.535,39.505,157.429
C03578=1038.468,78.140,409.681,169.533,39.504,157.429
C03579=1038.462,77.890,409.699,169.531,39.505,157.429
C03580=1038.455,77.641,409.718,169.529,39.504,157.429
C03581=1038.450,77.393,409.736,169.527,39.504,157.428
C03582=1038.442,77.107,409.757,169.525,39.504,157.428
C03583=1038.435,76.820,409.779,169.523,39.503,157.428
C03584=1038.428,76.535,409.799,169.519,39.503,157.428
C03585=1038.420,76.248,409.820,169.517,39.502,157.428
C03586=1038.414,75.999,409.839,169.515,39.503,157.428
C03587=1038.408,75.749,409.857,169.513,39.502,157.428
C03588=1038.401,75.500,409.876,169.511,39.502,157.428
C03589=1038.394,75.251,409.894,169.509,39.502,157.427
C03590=1038.389,75.002,409.911,169.507,39.501,157.427
C03591=1038.382,74.753,409.930,169.505,39.501,157.427
C03592=1038.376,74.503,409.948,169.504,39.501,157.427
C03593=1038.370,74.254,409.967,169.501,39.500,157.427
C03594=1038.364,74.005,409.985,169.499,39.500,157.427
C03595=1038.357,73.756,410.003,169.497,39.500,157.427
C03596=1038.351,73.506,410.022,169.495,39.500,157.427
C03597=1038.345,73.257,410.039,169.493,39.499,157.426
C03598=1038.339,73.008,410.058,169.491,39.499,157.426
C03599=1038.332,72.759,410.075,169.489,39.499,157.426
C03600=1038.326,72.510,410.094,169.487,39.498,157.426
C03601=1038.319,72.260,410.112,169.485,39.498,157.426
C03602=1038.313,72.011,410.131,169.482,39.498,157.426
C03603=1038.308,71.762,410.148,169.480,39.497,157.426
C03604=1038.301,71.513,410.167,169.478,39.498,157.426
C03605=1038.295,71.263,410.185,169.476,39.497,157.425
C03606=1038.289,71.014,410.203,169.474,39.497,157.425
C03607=1038.282,70.764,410.221,169.472,39.497,157.425
C03608=1038.276,70.516,410.239,169.471,39.496,157.425
C03609=1038.270,70.266,410.257,169.469,39.496,157.425
C03610=1038.263,70.017,410.276,169.467,39.496,157.425
C03611=1038.257,69.767,410.294,169.465,39.495,157.425
C03612=1038.252,69.518,410.311,169.462,39.495,157.425
C03613=1038.245,69.269,410.330,169.460,39.495,157.425
C03614=1038.238,69.020,410.347,169.458,39.495,157.424
C03615=1038.232,68.771,410.366,169.456,39.494,157.424
C03616=1038.226,68.521,410.384,169.454,39.494,157.424
C03617=1038.220,68.272,410.401,169.452,39.494,157.424
C03618=1038.213,68.023,410.419,169.450,39.494,157.424
C03619=1038.207,67.773,410.437,169.448,39.493,157.424
C03620=1038.201,67.524,410.455,169.446,39.493,157.424
C03621=1038.194,67.275,410.473,169.444,39.493,157.424
C03622=1038.188,67.026,410.491,169.441,39.493,157.423
C03623=1038.182,66.776,410.509,169.439,39.493,157.423
C03624=1038.176,66.527,410.527,169.438,39.492,157.423
C03625=1038.169,66.277,410.545,169.436,39.492,157.423
C03626=1038.163,66.028,410.562,169.434,39.492,157.423
C03627=1038.157,65.779,410.581,169.432,39.491,157.423
C03628=1038.150,65.530,410.598,169.430,39.492,157.423
C03629=1038.144,65.280,410.616,169.428,39.491,157.423
C03630=1038.138,65.031,410.634,169.426,39.491,157.423
C03631=1038.131,64.782,410.652,169.424,39.491,157.423
C03632=1038.125,64.532,410.670,169.421,39.490,157.422
C03633=1038.120,64.283,410.687,169.419,39.490,157.422
C03634=1038.113,64.034,410.705,169.417,39.490,157.422
C03635=1038.106,63.785,410.723,169.415,39.489,157.422
C03636=1038.099,63.535,410.741,169.413,39.490,157.422
C03637=1038.094,63.286,410.758,169.411,39.489,157.422
C03638=1038.087,63.037,410.776,169.409,39.489,157.422
